C08965=1019.841,-8.472,-102.051,166.453,52.235,159.485
C08966=1019.835,-8.722,-102.038,166.450,52.240,159.486
C08967=1019.829,-8.971,-102.024,166.447,52.245,159.486
C08968=1019.824,-9.221,-102.010,166.445,52.250,159.487
C08969=1019.818,-9.471,-101.998,166.442,52.256,159.487
C08970=1019.812,-9.720,-101.985,166.439,52.261,159.487
C08971=1019.806,-9.970,-101.971,166.436,52.266,159.488
C08972=1019.801,-10.219,-101.959,166.434,52.272,159.489
C08973=1019.796,-10.469,-101.945,166.431,52.277,159.489
C08974=1019.789,-10.718,-101.932,166.428,52.283,159.489
C08975=1019.784,-10.968,-101.918,166.425,52.288,159.490
C08976=1019.778,-11.218,-101.906,166.423,52.293,159.490
C08977=1019.772,-11.467,-101.892,166.420,52.298,159.491
C08978=1019.767,-11.717,-101.879,166.417,52.304,159.491
C08979=1019.760,-11.966,-101.866,166.414,52.309,159.491
C08980=1019.756,-12.216,-101.853,166.412,52.314,159.492
C08981=1019.750,-12.465,-101.840,166.408,52.319,159.492
C08982=1019.745,-12.715,-101.827,166.405,52.324,159.493
C08983=1019.738,-12.965,-101.814,166.403,52.331,159.493
C08984=1019.732,-13.215,-101.801,166.401,52.335,159.494
C08985=1019.727,-13.464,-101.787,166.398,52.341,159.494
C08986=1019.722,-13.713,-101.775,166.395,52.346,159.495
C08987=1019.716,-13.963,-101.761,166.393,52.351,159.495
C08988=1019.710,-14.213,-101.749,166.389,52.356,159.496
C08989=1019.704,-14.463,-101.736,166.386,52.362,159.496
C08990=1019.699,-14.712,-101.722,166.383,52.367,159.496
C08991=1019.694,-14.961,-101.710,166.381,52.372,159.497
C08992=1019.688,-15.211,-101.696,166.378,52.377,159.497
C08993=1019.682,-15.461,-101.684,166.375,52.383,159.498
C08994=1019.676,-15.710,-101.670,166.373,52.388,159.498
C08995=1019.671,-15.960,-101.657,166.370,52.393,159.499
C08996=1019.665,-16.209,-101.645,166.367,52.398,159.499
C08997=1019.660,-16.459,-101.632,166.364,52.404,159.499
C08998=1019.653,-16.709,-101.619,166.361,52.409,159.500
C08999=1019.647,-16.959,-101.607,166.359,52.414,159.500
C09000=1019.642,-17.209,-101.593,166.356,52.419,159.501
C09001=1019.637,-17.457,-101.580,166.353,52.425,159.501
C09002=1019.631,-17.707,-101.568,166.350,52.431,159.502
C09003=1019.625,-17.957,-101.555,166.347,52.436,159.502
C09004=1019.619,-18.207,-101.543,166.345,52.441,159.503
C09005=1019.614,-18.456,-101.531,166.342,52.446,159.503
C09006=1019.607,-18.705,-101.517,166.339,52.452,159.503
C09007=1019.602,-18.956,-101.504,166.336,52.457,159.504
C09008=1019.596,-19.205,-101.492,166.334,52.462,159.504
C09009=1019.591,-19.455,-101.479,166.331,52.467,159.505
C09010=1019.585,-19.705,-101.467,166.328,52.473,159.505
C09011=1019.579,-19.954,-101.454,166.325,52.479,159.506
C09012=1019.574,-20.203,-101.441,166.322,52.484,159.506
C09013=1019.568,-20.453,-101.429,166.320,52.489,159.507
C09014=1019.562,-20.703,-101.416,166.317,52.494,159.507
C09015=1019.556,-20.981,-101.402,166.314,52.500,159.507
C09016=1019.550,-21.259,-101.388,166.310,52.506,159.508
C09017=1019.543,-21.539,-101.373,166.307,52.512,159.509
C09018=1019.537,-21.817,-101.360,166.304,52.518,159.509
C09019=1019.531,-22.067,-101.347,166.301,52.523,159.509
C09020=1019.525,-22.316,-101.335,166.298,52.528,159.510
C09021=1019.520,-22.566,-101.322,166.295,52.534,159.510
C09022=1019.514,-22.816,-101.309,166.293,52.539,159.511
C09023=1019.509,-23.065,-101.297,166.290,52.544,159.511
C09024=1019.503,-23.315,-101.284,166.287,52.549,159.511
C09025=1019.497,-23.565,-101.271,166.284,52.555,159.512
C09026=1019.492,-23.814,-101.259,166.281,52.560,159.512
C09027=1019.486,-24.064,-101.246,166.279,52.565,159.513
C09028=1019.480,-24.314,-101.234,166.276,52.570,159.513
C09029=1019.475,-24.563,-101.221,166.273,52.576,159.514
C09030=1019.469,-24.813,-101.209,166.271,52.581,159.514
C09031=1019.464,-25.062,-101.196,166.268,52.586,159.514
C09032=1019.458,-25.312,-101.184,166.265,52.591,159.515
C09033=1019.452,-25.562,-101.171,166.262,52.597,159.515
C09034=1019.447,-25.811,-101.159,166.260,52.602,159.516
C09035=1019.441,-26.061,-101.147,166.256,52.606,159.516
C09036=1019.436,-26.310,-101.134,166.253,52.612,159.516
C09037=1019.430,-26.560,-101.122,166.250,52.617,159.517
C09038=1019.425,-26.810,-101.109,166.248,52.622,159.517
C09039=1019.419,-27.059,-101.096,166.245,52.628,159.518
C09040=1019.413,-27.309,-101.084,166.242,52.633,159.518
C09041=1019.408,-27.558,-101.072,166.239,52.638,159.518
C09042=1019.402,-27.808,-101.059,166.237,52.643,159.519
C09043=1019.397,-28.059,-101.047,166.234,52.649,159.519
C09044=1019.391,-28.308,-101.035,166.231,52.654,159.520
C09045=1019.385,-28.558,-101.023,166.228,52.659,159.520
C09046=1019.379,-28.807,-101.011,166.225,52.665,159.520
C09047=1019.373,-29.057,-100.998,166.223,52.670,159.521
C09048=1019.368,-29.306,-100.986,166.220,52.675,159.521
C09049=1019.363,-29.556,-100.974,166.217,52.680,159.522
C09050=1019.357,-29.806,-100.962,166.214,52.686,159.522
C09051=1019.351,-30.055,-100.950,166.211,52.691,159.523
C09052=1019.345,-30.305,-100.938,166.208,52.697,159.523
C09053=1019.340,-30.555,-100.926,166.206,52.702,159.523
C09054=1019.334,-30.805,-100.914,166.203,52.707,159.524
C09055=1019.328,-31.054,-100.902,166.200,52.712,159.524
C09056=1019.323,-31.304,-100.889,166.197,52.718,159.525
C09057=1019.317,-31.553,-100.878,166.193,52.723,159.525
C09058=1019.311,-31.803,-100.866,166.191,52.728,159.526
C09059=1019.306,-32.052,-100.853,166.188,52.733,159.526
C09060=1019.300,-32.302,-100.841,166.185,52.739,159.526
C09061=1019.295,-32.552,-100.829,166.182,52.744,159.527
C09062=1019.289,-32.802,-100.817,166.179,52.749,159.527
C09063=1019.283,-33.051,-100.805,166.177,52.755,159.528
C09064=1019.277,-33.301,-100.793,166.174,52.760,159.528
C09065=1019.272,-33.550,-100.781,166.171,52.765,159.528
C09066=1019.266,-33.800,-100.769,166.168,52.771,159.529
C09067=1019.261,-34.050,-100.757,166.165,52.775,159.529
C09068=1019.255,-34.299,-100.746,166.163,52.780,159.529
C09069=1019.249,-34.549,-100.733,166.160,52.786,159.530
C09070=1019.244,-34.799,-100.722,166.157,52.791,159.530
C09071=1019.238,-35.049,-100.709,166.154,52.796,159.531
C09072=1019.233,-35.298,-100.697,166.151,52.802,159.531
C09073=1019.228,-35.548,-100.685,166.149,52.807,159.531
C09074=1019.221,-35.797,-100.673,166.146,52.812,159.532
C09075=1019.216,-36.047,-100.662,166.143,52.818,159.532
C09076=1019.210,-36.297,-100.649,166.140,52.823,159.533
C09077=1019.205,-36.546,-100.637,166.136,52.828,159.533
C09078=1019.200,-36.796,-100.626,166.134,52.833,159.533
C09079=1019.193,-37.074,-100.612,166.130,52.839,159.534
C09080=1019.187,-37.352,-100.599,166.127,52.845,159.534
C09081=1019.181,-37.629,-100.586,166.124,52.850,159.535
C09082=1019.175,-37.908,-100.573,166.121,52.856,159.535
C09083=1019.169,-38.157,-100.560,166.119,52.861,159.536
C09084=1019.163,-38.406,-100.549,166.116,52.867,159.536
C09085=1019.158,-38.656,-100.537,166.112,52.871,159.536
C09086=1019.152,-38.905,-100.525,166.109,52.877,159.536
C09087=1019.147,-39.155,-100.513,166.107,52.882,159.537
C09088=1019.141,-39.405,-100.501,166.104,52.887,159.537
C09089=1019.136,-39.655,-100.490,166.101,52.893,159.538
C09090=1019.131,-39.904,-100.478,166.098,52.898,159.538
C09091=1019.124,-40.154,-100.466,166.095,52.903,159.539
C09092=1019.119,-40.404,-100.455,166.092,52.909,159.539
C09093=1019.113,-40.653,-100.444,166.089,52.914,159.539
C09094=1019.107,-40.903,-100.432,166.087,52.919,159.540
C09095=1019.102,-41.153,-100.421,166.084,52.925,159.540
C09096=1019.097,-41.402,-100.409,166.081,52.930,159.541
C09097=1019.090,-41.652,-100.397,166.078,52.935,159.541
C09098=1019.085,-41.902,-100.386,166.075,52.941,159.541
C09099=1019.079,-42.151,-100.375,166.072,52.946,159.542
C09100=1019.073,-42.401,-100.362,166.069,52.951,159.542
C09101=1019.068,-42.651,-100.351,166.066,52.956,159.542
C09102=1019.063,-42.900,-100.340,166.064,52.961,159.543
C09103=1019.057,-43.150,-100.328,166.061,52.967,159.543
C09104=1019.051,-43.400,-100.317,166.058,52.972,159.544
C09105=1019.046,-43.650,-100.305,166.055,52.978,159.544
C09106=1019.040,-43.899,-100.294,166.052,52.983,159.544
C09107=1019.034,-44.149,-100.282,166.049,52.988,159.545
C09108=1019.029,-44.399,-100.271,166.047,52.993,159.545
C09109=1019.024,-44.648,-100.259,166.044,52.999,159.546
C09110=1019.018,-44.898,-100.248,166.041,53.004,159.546
C09111=1019.012,-45.148,-100.236,166.037,53.009,159.546
C09112=1019.006,-45.397,-100.225,166.034,53.014,159.546
C09113=1019.001,-45.647,-100.214,166.031,53.020,159.547
C09114=1018.995,-45.896,-100.203,166.028,53.025,159.547
C09115=1018.990,-46.146,-100.190,166.026,53.030,159.548
C09116=1018.984,-46.396,-100.179,166.023,53.036,159.548
C09117=1018.979,-46.646,-100.168,166.020,53.041,159.549
C09118=1018.973,-46.895,-100.157,166.017,53.046,159.549
C09119=1018.968,-47.145,-100.145,166.014,53.051,159.549
C09120=1018.962,-47.394,-100.135,166.011,53.056,159.549
C09121=1018.956,-47.644,-100.122,166.009,53.061,159.550
C09122=1018.951,-47.894,-100.111,166.006,53.067,159.550
C09123=1018.946,-48.144,-100.100,166.003,53.072,159.551
C09124=1018.940,-48.393,-100.089,165.999,53.077,159.551
C09125=1018.935,-48.643,-100.077,165.996,53.082,159.551
C09126=1018.930,-48.893,-100.066,165.994,53.087,159.552
C09127=1018.924,-49.142,-100.055,165.991,53.093,159.552
C09128=1018.919,-49.393,-100.043,165.988,53.098,159.552
C09129=1018.913,-49.642,-100.031,165.985,53.103,159.553
C09130=1018.908,-49.891,-100.020,165.982,53.108,159.553
C09131=1018.902,-50.141,-100.009,165.979,53.114,159.553
C09132=1018.897,-50.391,-99.998,165.977,53.119,159.554
C09133=1018.891,-50.640,-99.987,165.974,53.124,159.554
C09134=1018.886,-50.890,-99.975,165.970,53.129,159.554
C09135=1018.880,-51.140,-99.964,165.967,53.134,159.555
C09136=1018.874,-51.390,-99.953,165.964,53.140,159.555
C09137=1018.868,-51.639,-99.942,165.961,53.145,159.556
C09138=1018.863,-51.889,-99.932,165.958,53.151,159.556
C09139=1018.857,-52.139,-99.921,165.955,53.156,159.556
C09140=1018.851,-52.388,-99.910,165.952,53.161,159.557
C09141=1018.846,-52.638,-99.899,165.949,53.167,159.557
C09142=1018.841,-52.887,-99.888,165.946,53.172,159.557
C09143=1018.834,-53.165,-99.876,165.944,53.178,159.558
C09144=1018.827,-53.444,-99.864,165.940,53.185,159.558
C09145=1018.821,-53.722,-99.852,165.937,53.190,159.559
C09146=1018.815,-54.000,-99.840,165.934,53.197,159.559
C09147=1018.809,-54.250,-99.829,165.931,53.202,159.560
///RCONF 1,0,0,1,0,0,0,0,0,0,0,0,0,0,0,0,0,0,0,0,0,0,0,0
C09148=1018.804,-54.499,-99.818,165.928,53.208,159.560
C09149=1018.798,-54.749,-99.808,165.925,53.213,159.560
C09150=1018.792,-54.999,-99.797,165.922,53.219,159.561
C09151=1018.787,-55.248,-99.786,165.919,53.224,159.561
C09152=1018.782,-55.498,-99.775,165.916,53.229,159.562
C09153=1018.776,-55.748,-99.765,165.914,53.235,159.562
C09154=1018.770,-55.998,-99.754,165.911,53.240,159.562
C09155=1018.765,-56.247,-99.743,165.908,53.245,159.563
C09156=1018.759,-56.497,-99.732,165.905,53.251,159.563
C09157=1018.754,-56.747,-99.722,165.901,53.256,159.563
C09158=1018.748,-56.996,-99.711,165.898,53.261,159.564
C09159=1018.742,-57.246,-99.700,165.895,53.266,159.564
C09160=1018.737,-57.496,-99.690,165.892,53.272,159.564
C09161=1018.731,-57.745,-99.679,165.889,53.277,159.565
C09162=1018.726,-57.995,-99.668,165.886,53.283,159.565
C09163=1018.720,-58.245,-99.657,165.883,53.288,159.566
C09164=1018.715,-58.495,-99.647,165.880,53.294,159.566
C09165=1018.709,-58.744,-99.636,165.877,53.299,159.566
C09166=1018.704,-58.994,-99.626,165.874,53.304,159.567
C09167=1018.698,-59.244,-99.615,165.871,53.310,159.567
C09168=1018.692,-59.493,-99.604,165.868,53.315,159.567
C09169=1018.687,-59.743,-99.594,165.865,53.320,159.568
C09170=1018.681,-59.993,-99.583,165.863,53.325,159.568
C09171=1018.675,-60.243,-99.573,165.860,53.331,159.568
C09172=1018.670,-60.493,-99.562,165.857,53.336,159.569
C09173=1018.665,-60.741,-99.551,165.854,53.341,159.569
C09174=1018.660,-60.992,-99.540,165.851,53.347,159.570
C09175=1018.654,-61.241,-99.530,165.848,53.352,159.570
C09176=1018.649,-61.491,-99.519,165.845,53.357,159.570
C09177=1018.643,-61.741,-99.509,165.842,53.363,159.570
C09178=1018.637,-61.990,-99.498,165.839,53.368,159.571
C09179=1018.632,-62.240,-99.487,165.836,53.373,159.571
C09180=1018.626,-62.490,-99.477,165.833,53.379,159.571
C09181=1018.621,-62.740,-99.466,165.830,53.384,159.572
C09182=1018.615,-62.989,-99.456,165.827,53.389,159.572
C09183=1018.610,-63.239,-99.446,165.824,53.394,159.573
C09184=1018.604,-63.488,-99.435,165.821,53.400,159.573
C09185=1018.599,-63.739,-99.425,165.818,53.405,159.573
C09186=1018.593,-63.988,-99.414,165.815,53.410,159.574
C09187=1018.588,-64.238,-99.404,165.812,53.416,159.574
C09188=1018.583,-64.488,-99.392,165.809,53.421,159.574
C09189=1018.578,-64.737,-99.382,165.806,53.426,159.574
C09190=1018.572,-64.987,-99.372,165.803,53.432,159.575
C09191=1018.567,-65.237,-99.361,165.800,53.437,159.575
C09192=1018.561,-65.487,-99.351,165.798,53.441,159.576
C09193=1018.556,-65.737,-99.340,165.795,53.447,159.576
C09194=1018.551,-65.986,-99.331,165.792,53.452,159.576
C09195=1018.545,-66.235,-99.320,165.789,53.458,159.577
C09196=1018.540,-66.486,-99.310,165.785,53.462,159.577
C09197=1018.534,-66.735,-99.299,165.782,53.468,159.577
C09198=1018.528,-66.985,-99.288,165.779,53.473,159.577
C09199=1018.524,-67.235,-99.279,165.776,53.479,159.578
C09200=1018.518,-67.484,-99.268,165.774,53.483,159.578
C09201=1018.512,-67.734,-99.258,165.771,53.489,159.579
C09202=1018.507,-67.984,-99.247,165.768,53.494,159.579
C09203=1018.502,-68.233,-99.237,165.765,53.499,159.579
C09204=1018.496,-68.483,-99.227,165.762,53.504,159.579
C09205=1018.491,-68.733,-99.215,165.759,53.510,159.580
C09206=1018.486,-68.983,-99.205,165.756,53.515,159.580
C09207=1018.479,-69.286,-99.193,165.752,53.521,159.580
C09208=1018.473,-69.590,-99.180,165.748,53.528,159.581
C09209=1018.466,-69.893,-99.168,165.746,53.534,159.581
C09210=1018.460,-70.196,-99.156,165.742,53.540,159.582
C09211=1018.455,-70.446,-99.145,165.739,53.545,159.582
C09212=1018.449,-70.696,-99.134,165.736,53.551,159.582
C09213=1018.445,-70.945,-99.125,165.732,53.555,159.582
C09214=1018.439,-71.196,-99.114,165.729,53.561,159.583
C09215=1018.433,-71.445,-99.104,165.726,53.566,159.583
C09216=1018.429,-71.694,-99.094,165.724,53.571,159.583
C09217=1018.423,-71.945,-99.084,165.721,53.576,159.584
C09218=1018.418,-72.195,-99.073,165.718,53.582,159.584
C09219=1018.413,-72.443,-99.063,165.715,53.586,159.584
C09220=1018.407,-72.694,-99.053,165.712,53.592,159.585
C09221=1018.402,-72.944,-99.043,165.708,53.597,159.585
C09222=1018.397,-73.193,-99.033,165.706,53.602,159.585
C09223=1018.391,-73.443,-99.022,165.703,53.607,159.586
C09224=1018.386,-73.693,-99.012,165.700,53.612,159.586
C09225=1018.381,-73.942,-99.002,165.697,53.617,159.586
C09226=1018.375,-74.192,-98.992,165.693,53.622,159.586
C09227=1018.370,-74.442,-98.982,165.691,53.628,159.587
C09228=1018.365,-74.692,-98.972,165.688,53.633,159.587
C09229=1018.360,-74.942,-98.962,165.685,53.639,159.587
C09230=1018.354,-75.191,-98.953,165.682,53.643,159.588
C09231=1018.349,-75.441,-98.942,165.679,53.648,159.588
C09232=1018.343,-75.691,-98.932,165.676,53.654,159.588
C09233=1018.338,-75.941,-98.922,165.673,53.659,159.589
C09234=1018.332,-76.190,-98.913,165.670,53.665,159.589
C09235=1018.327,-76.440,-98.903,165.667,53.670,159.589
C09236=1018.322,-76.690,-98.893,165.664,53.675,159.590
C09237=1018.316,-76.940,-98.883,165.661,53.681,159.590
C09238=1018.311,-77.189,-98.874,165.658,53.686,159.590
C09239=1018.306,-77.439,-98.863,165.655,53.691,159.590
C09240=1018.301,-77.689,-98.854,165.652,53.696,159.591
C09241=1018.295,-77.938,-98.844,165.649,53.702,159.591
C09242=1018.290,-78.188,-98.834,165.646,53.707,159.591
C09243=1018.285,-78.426,-98.825,165.643,53.712,159.592
C09244=1018.280,-78.663,-98.816,165.641,53.717,159.592
C09245=1018.275,-78.901,-98.806,165.637,53.722,159.592
C09246=1018.269,-79.139,-98.797,165.634,53.727,159.593
C09247=1018.264,-79.376,-98.788,165.632,53.732,159.593
C09248=1018.259,-79.614,-98.779,165.629,53.737,159.593
C09249=1018.254,-79.851,-98.769,165.625,53.742,159.593
C09250=1018.249,-80.089,-98.759,165.624,53.747,159.594
C09251=1018.244,-80.339,-98.751,165.620,53.752,159.594
C09252=1018.239,-80.589,-98.741,165.617,53.757,159.594
C09253=1018.233,-80.838,-98.731,165.614,53.763,159.595
C09254=1018.228,-81.088,-98.721,165.611,53.768,159.595
C09255=1018.222,-81.338,-98.713,165.608,53.774,159.595
C09256=1018.217,-81.588,-98.703,165.605,53.779,159.596
C09257=1018.211,-81.837,-98.693,165.602,53.785,159.596
C09258=1018.205,-82.088,-98.685,165.599,53.790,159.597
C09259=1018.201,-82.337,-98.675,165.597,53.796,159.597
C09260=1018.194,-82.587,-98.665,165.593,53.801,159.597
C09261=1018.190,-82.837,-98.656,165.590,53.806,159.597
C09262=1018.184,-83.087,-98.647,165.587,53.812,159.598
C09263=1018.179,-83.336,-98.637,165.584,53.817,159.598
C09264=1018.173,-83.586,-98.628,165.581,53.823,159.598
C09265=1018.168,-83.836,-98.618,165.578,53.828,159.599
C09266=1018.163,-84.085,-98.609,165.575,53.834,159.599
C09267=1018.157,-84.335,-98.600,165.572,53.838,159.599
C09268=1018.152,-84.585,-98.590,165.569,53.844,159.600
C09269=1018.146,-84.835,-98.581,165.566,53.849,159.600
C09270=1018.141,-85.085,-98.572,165.563,53.855,159.600
C09271=1018.135,-85.366,-98.561,165.559,53.861,159.600
C09272=1018.129,-85.647,-98.551,165.556,53.867,159.601
C09273=1018.122,-85.928,-98.540,165.553,53.873,159.601
C09274=1018.117,-86.209,-98.530,165.549,53.879,159.602
C09275=1018.111,-86.459,-98.521,165.546,53.884,159.602
C09276=1018.106,-86.709,-98.511,165.543,53.890,159.602
C09277=1018.101,-86.958,-98.503,165.540,53.895,159.603
C09278=1018.096,-87.208,-98.492,165.537,53.901,159.603
C09279=1018.090,-87.458,-98.484,165.534,53.906,159.603
C09280=1018.086,-87.708,-98.474,165.531,53.911,159.603
C09281=1018.080,-87.958,-98.465,165.528,53.917,159.604
C09282=1018.075,-88.207,-98.455,165.525,53.922,159.604
C09283=1018.070,-88.457,-98.447,165.522,53.928,159.604
C09284=1018.063,-88.707,-98.437,165.518,53.932,159.605
C09285=1018.059,-88.957,-98.428,165.515,53.938,159.605
C09286=1018.053,-89.206,-98.419,165.513,53.943,159.605
C09287=1018.048,-89.457,-98.410,165.510,53.949,159.606
C09288=1018.043,-89.706,-98.400,165.506,53.954,159.606
C09289=1018.037,-89.956,-98.392,165.503,53.959,159.606
C09290=1018.032,-90.206,-98.382,165.500,53.965,159.606
C09291=1018.027,-90.455,-98.373,165.498,53.969,159.607
C09292=1018.022,-90.705,-98.364,165.495,53.975,159.607
C09293=1018.017,-90.954,-98.355,165.492,53.980,159.607
C09294=1018.012,-91.205,-98.346,165.489,53.986,159.608
C09295=1018.006,-91.454,-98.336,165.486,53.990,159.608
C09296=1018.001,-91.704,-98.328,165.483,53.996,159.608
C09297=1017.996,-91.953,-98.318,165.480,54.001,159.609
C09298=1017.990,-92.204,-98.309,165.477,54.006,159.609
C09299=1017.985,-92.454,-98.300,165.474,54.012,159.609
C09300=1017.980,-92.703,-98.291,165.471,54.017,159.609
C09301=1017.975,-92.953,-98.283,165.467,54.022,159.609
C09302=1017.970,-93.203,-98.273,165.464,54.028,159.610
C09303=1017.964,-93.453,-98.264,165.461,54.033,159.610
C09304=1017.959,-93.703,-98.255,165.458,54.038,159.610
C09305=1017.954,-93.952,-98.246,165.455,54.043,159.611
C09306=1017.949,-94.201,-98.237,165.452,54.049,159.611
C09307=1017.944,-94.451,-98.228,165.450,54.053,159.611
C09308=1017.938,-94.702,-98.219,165.447,54.059,159.612
C09309=1017.933,-94.951,-98.209,165.444,54.064,159.612
C09310=1017.928,-95.201,-98.201,165.441,54.069,159.612
C09311=1017.923,-95.451,-98.192,165.438,54.075,159.612
C09312=1017.918,-95.701,-98.183,165.434,54.080,159.613
C09313=1017.913,-95.950,-98.174,165.431,54.085,159.613
C09314=1017.908,-96.200,-98.165,165.428,54.091,159.613
C09315=1017.902,-96.450,-98.156,165.425,54.095,159.613
C09316=1017.897,-96.700,-98.148,165.422,54.101,159.614
C09317=1017.892,-96.949,-98.138,165.420,54.105,159.614
C09318=1017.887,-97.199,-98.129,165.417,54.111,159.614
C09319=1017.882,-97.449,-98.120,165.414,54.116,159.615
C09320=1017.877,-97.699,-98.112,165.411,54.121,159.615
C09321=1017.871,-97.949,-98.103,165.408,54.127,159.615
C09322=1017.867,-98.199,-98.094,165.405,54.132,159.615
C09323=1017.861,-98.448,-98.085,165.401,54.137,159.616
C09324=1017.856,-98.698,-98.076,165.398,54.143,159.616
C09325=1017.851,-98.948,-98.068,165.395,54.148,159.616
C09326=1017.845,-99.197,-98.059,165.393,54.154,159.617
C09327=1017.840,-99.447,-98.051,165.390,54.159,159.617
C09328=1017.835,-99.697,-98.042,165.386,54.164,159.617
C09329=1017.830,-99.947,-98.034,165.383,54.170,159.617
C09330=1017.825,-100.197,-98.025,165.380,54.175,159.618
C09331=1017.820,-100.446,-98.016,165.378,54.181,159.618
C09332=1017.815,-100.696,-98.008,165.374,54.186,159.618
C09333=1017.809,-100.946,-97.999,165.371,54.191,159.619
C09334=1017.803,-101.196,-97.990,165.368,54.197,159.619
C09335=1017.798,-101.479,-97.981,165.364,54.203,159.619
C09336=1017.792,-101.763,-97.971,165.362,54.209,159.620
C09337=1017.786,-102.046,-97.961,165.358,54.215,159.620
C09338=1017.780,-102.329,-97.952,165.354,54.221,159.620
C09339=1017.776,-102.579,-97.943,165.351,54.226,159.620
C09340=1017.771,-102.829,-97.935,165.348,54.232,159.621
C09341=1017.765,-103.079,-97.927,165.346,54.236,159.621
C09342=1017.760,-103.328,-97.918,165.343,54.242,159.621
C09343=1017.755,-103.578,-97.910,165.340,54.247,159.622
C09344=1017.750,-103.828,-97.901,165.337,54.252,159.622
C09345=1017.744,-104.078,-97.893,165.334,54.258,159.622
C09346=1017.739,-104.327,-97.884,165.331,54.263,159.622
C09347=1017.734,-104.577,-97.876,165.328,54.269,159.623
C09348=1017.728,-104.827,-97.867,165.324,54.274,159.623
C09349=1017.723,-105.077,-97.860,165.322,54.279,159.623
C09350=1017.718,-105.327,-97.851,165.319,54.285,159.624
C09351=1017.714,-105.577,-97.842,165.315,54.289,159.624
C09352=1017.708,-105.826,-97.834,165.312,54.295,159.624
C09353=1017.703,-106.076,-97.825,165.309,54.301,159.624
C09354=1017.698,-106.327,-97.817,165.306,54.305,159.624
C09355=1017.693,-106.576,-97.809,165.303,54.311,159.625
C09356=1017.688,-106.826,-97.800,165.300,54.316,159.625
C09357=1017.682,-107.076,-97.792,165.297,54.321,159.625
C09358=1017.678,-107.325,-97.784,165.294,54.327,159.626
C09359=1017.673,-107.575,-97.776,165.291,54.332,159.626
C09360=1017.668,-107.825,-97.768,165.288,54.337,159.626
C09361=1017.662,-108.074,-97.759,165.285,54.343,159.626
C09362=1017.657,-108.325,-97.751,165.282,54.348,159.627
C09363=1017.652,-108.575,-97.743,165.279,54.354,159.627
C09364=1017.647,-108.824,-97.734,165.276,54.359,159.627
C09365=1017.641,-109.074,-97.727,165.273,54.364,159.627
C09366=1017.636,-109.324,-97.719,165.270,54.370,159.628
C09367=1017.631,-109.573,-97.711,165.267,54.375,159.628
C09368=1017.626,-109.823,-97.703,165.264,54.380,159.628
C09369=1017.621,-110.073,-97.694,165.261,54.386,159.629
C09370=1017.616,-110.323,-97.687,165.258,54.391,159.629
C09371=1017.611,-110.573,-97.678,165.254,54.396,159.629
C09372=1017.605,-110.823,-97.670,165.253,54.401,159.629
C09373=1017.601,-111.072,-97.662,165.250,54.407,159.630
C09374=1017.595,-111.322,-97.654,165.247,54.413,159.630
C09375=1017.590,-111.572,-97.647,165.243,54.417,159.630
C09376=1017.585,-111.822,-97.638,165.240,54.423,159.631
C09377=1017.580,-112.072,-97.630,165.238,54.428,159.631
C09378=1017.575,-112.321,-97.622,165.234,54.433,159.631
C09379=1017.570,-112.571,-97.614,165.231,54.439,159.631
C09380=1017.565,-112.821,-97.606,165.228,54.444,159.632
C09381=1017.560,-113.071,-97.597,165.225,54.449,159.632
C09382=1017.555,-113.321,-97.590,165.222,54.455,159.632
C09383=1017.549,-113.570,-97.582,165.219,54.460,159.632
C09384=1017.544,-113.820,-97.574,165.216,54.465,159.633
C09385=1017.539,-114.070,-97.566,165.213,54.471,159.633
C09386=1017.534,-114.320,-97.558,165.210,54.476,159.633
C09387=1017.530,-114.569,-97.550,165.207,54.481,159.633
C09388=1017.525,-114.820,-97.542,165.204,54.487,159.634
C09389=1017.519,-115.070,-97.535,165.201,54.492,159.634
C09390=1017.514,-115.319,-97.527,165.198,54.497,159.634
C09391=1017.509,-115.569,-97.519,165.195,54.503,159.634
C09392=1017.504,-115.819,-97.511,165.192,54.508,159.635
C09393=1017.498,-116.069,-97.503,165.188,54.513,159.635
C09394=1017.494,-116.319,-97.496,165.186,54.519,159.635
C09395=1017.489,-116.568,-97.488,165.183,54.524,159.636
C09396=1017.484,-116.819,-97.480,165.181,54.530,159.636
C09397=1017.479,-117.068,-97.472,165.177,54.534,159.636
C09398=1017.473,-117.318,-97.465,165.175,54.540,159.636
C09399=1017.468,-117.601,-97.456,165.171,54.546,159.637
C09400=1017.462,-117.885,-97.447,165.167,54.553,159.637
C09401=1017.457,-118.168,-97.438,165.164,54.558,159.637
C09402=1017.451,-118.451,-97.429,165.160,54.564,159.637
C09403=1017.446,-118.701,-97.422,165.157,54.570,159.638
C09404=1017.440,-118.951,-97.414,165.155,54.575,159.638
C09405=1017.435,-119.200,-97.406,165.151,54.580,159.638
C09406=1017.430,-119.451,-97.399,165.148,54.586,159.639
C09407=1017.425,-119.700,-97.392,165.145,54.591,159.639
C09408=1017.420,-119.950,-97.384,165.142,54.596,159.639
C09409=1017.415,-120.201,-97.376,165.139,54.602,159.639
C09410=1017.411,-120.450,-97.368,165.137,54.607,159.640
C09411=1017.405,-120.700,-97.361,165.134,54.612,159.640
C09412=1017.400,-120.950,-97.353,165.131,54.618,159.640
C09413=1017.396,-121.200,-97.346,165.128,54.623,159.641
C09414=1017.390,-121.450,-97.339,165.125,54.628,159.641
C09415=1017.385,-121.699,-97.330,165.122,54.634,159.641
C09416=1017.380,-121.949,-97.323,165.119,54.639,159.641
C09417=1017.375,-122.198,-97.316,165.116,54.644,159.641
C09418=1017.370,-122.449,-97.308,165.113,54.650,159.642
C09419=1017.365,-122.699,-97.300,165.110,54.655,159.642
C09420=1017.360,-122.948,-97.294,165.107,54.660,159.642
C09421=1017.355,-123.199,-97.286,165.104,54.666,159.643
C09422=1017.350,-123.447,-97.278,165.100,54.670,159.643
C09423=1017.345,-123.698,-97.270,165.098,54.676,159.643
C09424=1017.341,-123.947,-97.263,165.095,54.682,159.643
C09425=1017.335,-124.197,-97.256,165.092,54.686,159.644
C09426=1017.331,-124.447,-97.249,165.090,54.692,159.644
C09427=1017.326,-124.697,-97.241,165.087,54.697,159.644
C09428=1017.321,-124.947,-97.234,165.083,54.702,159.644
C09429=1017.316,-125.197,-97.226,165.080,54.708,159.645
C09430=1017.311,-125.446,-97.219,165.078,54.713,159.645
C09431=1017.306,-125.697,-97.212,165.074,54.718,159.645
C09432=1017.300,-125.946,-97.205,165.071,54.724,159.645
C09433=1017.296,-126.196,-97.197,165.068,54.729,159.646
C09434=1017.290,-126.446,-97.190,165.065,54.734,159.646
C09435=1017.285,-126.696,-97.182,165.062,54.740,159.646
C09436=1017.280,-126.945,-97.176,165.059,54.746,159.646
C09437=1017.275,-127.196,-97.168,165.056,54.750,159.646
C09438=1017.270,-127.445,-97.161,165.053,54.756,159.647
C09439=1017.266,-127.694,-97.154,165.050,54.762,159.647
C09440=1017.260,-127.944,-97.146,165.047,54.766,159.647
C09441=1017.256,-128.194,-97.139,165.045,54.772,159.648
C09442=1017.252,-128.444,-97.132,165.042,54.777,159.648
C09443=1017.248,-128.693,-97.123,165.039,54.780,159.648
C09444=1017.244,-128.942,-97.114,165.036,54.784,159.648
C09445=1017.240,-129.193,-97.105,165.033,54.787,159.648
C09446=1017.237,-129.442,-97.094,165.031,54.790,159.648
C09447=1017.235,-129.692,-97.083,165.028,54.792,159.647
C09448=1017.233,-129.941,-97.072,165.026,54.793,159.647
C09449=1017.231,-130.191,-97.060,165.023,54.794,159.646
C09450=1017.230,-130.441,-97.047,165.021,54.794,159.646
C09451=1017.229,-130.690,-97.034,165.019,54.794,159.646
C09452=1017.229,-130.940,-97.020,165.017,54.793,159.645
C09453=1017.229,-131.190,-97.006,165.014,54.791,159.644
C09454=1017.229,-131.439,-96.991,165.012,54.789,159.643
C09455=1017.230,-131.689,-96.975,165.010,54.787,159.642
C09456=1017.231,-131.938,-96.959,165.008,54.784,159.641
C09457=1017.233,-132.189,-96.943,165.006,54.780,159.640
C09458=1017.235,-132.438,-96.924,165.005,54.776,159.639
C09459=1017.237,-132.688,-96.907,165.003,54.771,159.638
C09460=1017.240,-132.938,-96.888,165.000,54.766,159.636
C09461=1017.243,-133.188,-96.869,164.999,54.760,159.635
C09462=1017.247,-133.437,-96.850,164.997,54.753,159.634
C09463=1016.989,-133.463,-97.235,164.957,55.109,159.686
C09464=1016.985,-133.214,-97.254,164.959,55.115,159.688
C09465=1016.982,-132.964,-97.273,164.960,55.121,159.689
C09466=1016.980,-132.715,-97.292,164.962,55.126,159.691
C09467=1016.977,-132.464,-97.310,164.964,55.131,159.692
C09468=1016.975,-132.215,-97.327,164.966,55.135,159.693
C09469=1016.974,-131.965,-97.344,164.968,55.139,159.694
C09470=1016.972,-131.715,-97.361,164.970,55.142,159.695
C09471=1016.971,-131.466,-97.377,164.972,55.145,159.696
C09472=1016.971,-131.216,-97.392,164.974,55.147,159.697
C09473=1016.971,-130.967,-97.406,164.976,55.148,159.698
C09474=1016.971,-130.717,-97.420,164.979,55.149,159.699
C09475=1016.972,-130.467,-97.433,164.980,55.149,159.699
C09476=1016.974,-130.218,-97.445,164.983,55.149,159.700
C09477=1016.975,-129.968,-97.457,164.985,55.148,159.700
C09478=1016.977,-129.718,-97.468,164.988,55.146,159.700
C09479=1016.979,-129.468,-97.480,164.991,55.144,159.701
C09480=1016.982,-129.219,-97.490,164.993,55.142,159.701
C09481=1016.985,-128.969,-97.500,164.996,55.139,159.701
C09482=1016.989,-128.719,-97.509,164.999,55.135,159.701
C09483=1016.993,-128.470,-97.517,165.002,55.131,159.701
C09484=1016.998,-128.220,-97.525,165.004,55.127,159.701
C09485=1017.002,-127.971,-97.532,165.007,55.121,159.700
C09486=1017.007,-127.722,-97.539,165.010,55.116,159.700
C09487=1017.012,-127.471,-97.547,165.013,55.111,159.700
C09488=1017.017,-127.222,-97.554,165.016,55.105,159.699
C09489=1017.022,-126.972,-97.561,165.018,55.099,159.699
C09490=1017.027,-126.722,-97.568,165.022,55.094,159.699
C09491=1017.032,-126.473,-97.576,165.025,55.089,159.699
C09492=1017.037,-126.223,-97.583,165.027,55.083,159.698
C09493=1017.042,-125.973,-97.590,165.030,55.077,159.698
C09494=1017.047,-125.723,-97.597,165.034,55.073,159.698
C09495=1017.051,-125.473,-97.604,165.036,55.067,159.698
C09496=1017.057,-125.223,-97.611,165.039,55.061,159.697
C09497=1017.061,-124.973,-97.619,165.042,55.056,159.697
C09498=1017.067,-124.723,-97.626,165.045,55.051,159.697
C09499=1017.072,-124.473,-97.633,165.048,55.045,159.697
C09500=1017.076,-124.223,-97.641,165.051,55.039,159.696
C09501=1017.082,-123.974,-97.648,165.054,55.034,159.696
C09502=1017.087,-123.723,-97.655,165.057,55.029,159.696
C09503=1017.091,-123.474,-97.664,165.060,55.023,159.695
C09504=1017.097,-123.224,-97.671,165.063,55.018,159.695
C09505=1017.101,-122.975,-97.678,165.066,55.013,159.695
C09506=1017.106,-122.724,-97.686,165.069,55.007,159.695
C09507=1017.111,-122.475,-97.693,165.072,55.002,159.694
C09508=1017.116,-122.225,-97.701,165.075,54.996,159.694
C09509=1017.121,-121.975,-97.707,165.078,54.991,159.694
C09510=1017.126,-121.725,-97.715,165.081,54.985,159.694
C09511=1017.131,-121.475,-97.723,165.084,54.980,159.693
C09512=1017.136,-121.225,-97.730,165.087,54.974,159.693
C09513=1017.141,-120.976,-97.738,165.090,54.969,159.693
C09514=1017.146,-120.726,-97.746,165.093,54.964,159.693
C09515=1017.151,-120.476,-97.753,165.096,54.958,159.692
C09516=1017.156,-120.226,-97.760,165.098,54.952,159.692
C09517=1017.161,-119.976,-97.768,165.102,54.948,159.692
C09518=1017.166,-119.727,-97.776,165.105,54.942,159.691
C09519=1017.171,-119.477,-97.783,165.107,54.936,159.691
C09520=1017.176,-119.227,-97.791,165.110,54.931,159.691
C09521=1017.181,-118.977,-97.798,165.114,54.926,159.691
C09522=1017.186,-118.727,-97.806,165.116,54.920,159.690
C09523=1017.191,-118.478,-97.814,165.119,54.915,159.690
C09524=1017.197,-118.194,-97.822,165.123,54.909,159.690
C09525=1017.203,-117.911,-97.831,165.127,54.902,159.689
C09526=1017.208,-117.628,-97.839,165.130,54.896,159.689
C09527=1017.214,-117.345,-97.849,165.133,54.889,159.689
C09528=1017.219,-117.095,-97.856,165.136,54.885,159.689
C09529=1017.224,-116.845,-97.863,165.139,54.879,159.688
C09530=1017.229,-116.595,-97.872,165.142,54.873,159.688
C09531=1017.234,-116.345,-97.880,165.145,54.868,159.688
C09532=1017.239,-116.096,-97.886,165.148,54.863,159.687
C09533=1017.244,-115.846,-97.895,165.151,54.857,159.687
C09534=1017.249,-115.596,-97.903,165.154,54.852,159.687
C09535=1017.254,-115.346,-97.910,165.158,54.846,159.687
C09536=1017.260,-115.097,-97.918,165.160,54.840,159.686
C09537=1017.265,-114.846,-97.926,165.164,54.835,159.686
C09538=1017.270,-114.596,-97.934,165.167,54.830,159.686
C09539=1017.274,-114.347,-97.942,165.169,54.824,159.686
C09540=1017.279,-114.097,-97.949,165.172,54.818,159.685
C09541=1017.284,-113.847,-97.958,165.176,54.813,159.685
C09542=1017.290,-113.598,-97.965,165.178,54.808,159.685
C09543=1017.295,-113.348,-97.973,165.181,54.802,159.684
C09544=1017.300,-113.098,-97.981,165.184,54.797,159.684
C09545=1017.305,-112.848,-97.989,165.188,54.792,159.684
C09546=1017.309,-112.598,-97.997,165.190,54.786,159.684
C09547=1017.315,-112.348,-98.005,165.193,54.781,159.683
C09548=1017.320,-112.098,-98.013,165.196,54.775,159.683
C09549=1017.325,-111.848,-98.022,165.199,54.769,159.683
C09550=1017.330,-111.599,-98.028,165.202,54.765,159.683
C09551=1017.335,-111.349,-98.037,165.205,54.759,159.682
C09552=1017.340,-111.099,-98.045,165.208,54.753,159.682
C09553=1017.345,-110.849,-98.053,165.211,54.748,159.681
C09554=1017.350,-110.599,-98.061,165.214,54.742,159.681
C09555=1017.355,-110.350,-98.069,165.217,54.737,159.681
C09556=1017.360,-110.100,-98.077,165.220,54.732,159.681
C09557=1017.365,-109.850,-98.085,165.223,54.726,159.680
C09558=1017.371,-109.600,-98.094,165.226,54.720,159.680
C09559=1017.376,-109.350,-98.101,165.228,54.715,159.680
C09560=1017.381,-109.101,-98.109,165.232,54.710,159.680
C09561=1017.386,-108.851,-98.117,165.235,54.704,159.679
C09562=1017.391,-108.601,-98.125,165.239,54.698,159.679
C09563=1017.396,-108.351,-98.134,165.241,54.693,159.679
C09564=1017.401,-108.101,-98.142,165.244,54.687,159.678
C09565=1017.407,-107.851,-98.150,165.247,54.682,159.678
C09566=1017.412,-107.602,-98.159,165.250,54.677,159.678
C09567=1017.416,-107.352,-98.166,165.253,54.671,159.678
C09568=1017.421,-107.102,-98.174,165.256,54.666,159.677
C09569=1017.427,-106.853,-98.183,165.259,54.660,159.677
C09570=1017.432,-106.603,-98.191,165.262,54.654,159.677
C09571=1017.437,-106.353,-98.199,165.265,54.650,159.676
C09572=1017.442,-106.103,-98.208,165.268,54.644,159.676
C09573=1017.448,-105.853,-98.216,165.271,54.638,159.676
C09574=1017.453,-105.603,-98.225,165.274,54.633,159.675
C09575=1017.458,-105.353,-98.232,165.277,54.628,159.675
C09576=1017.463,-105.103,-98.241,165.280,54.622,159.675
C09577=1017.468,-104.854,-98.249,165.283,54.617,159.675
C09578=1017.473,-104.605,-98.257,165.286,54.611,159.674
C09579=1017.477,-104.355,-98.267,165.289,54.606,159.674
C09580=1017.482,-104.104,-98.274,165.292,54.601,159.674
C09581=1017.488,-103.855,-98.283,165.295,54.595,159.673
C09582=1017.493,-103.605,-98.291,165.298,54.590,159.673
C09583=1017.498,-103.355,-98.300,165.301,54.584,159.673
C09584=1017.503,-103.105,-98.308,165.304,54.579,159.673
C09585=1017.509,-102.856,-98.317,165.307,54.574,159.672
C09586=1017.514,-102.606,-98.325,165.310,54.568,159.672
C09587=1017.519,-102.356,-98.334,165.313,54.562,159.672
C09588=1017.525,-102.073,-98.343,165.316,54.557,159.671
C09589=1017.531,-101.790,-98.353,165.320,54.550,159.671
C09590=1017.537,-101.506,-98.363,165.324,54.544,159.671
C09591=1017.542,-101.224,-98.373,165.326,54.538,159.670
C09592=1017.547,-100.974,-98.381,165.329,54.532,159.670
C09593=1017.552,-100.723,-98.389,165.332,54.527,159.670
C09594=1017.557,-100.474,-98.397,165.336,54.521,159.670
C09595=1017.563,-100.224,-98.406,165.339,54.516,159.669
C09596=1017.568,-99.974,-98.414,165.342,54.510,159.669
C09597=1017.573,-99.725,-98.423,165.345,54.504,159.669
C09598=1017.578,-99.475,-98.431,165.348,54.499,159.668
C09599=1017.584,-99.225,-98.440,165.351,54.493,159.668
C09600=1017.588,-98.975,-98.449,165.354,54.488,159.668
C09601=1017.594,-98.725,-98.458,165.357,54.483,159.667
C09602=1017.599,-98.475,-98.466,165.360,54.477,159.667
C09603=1017.605,-98.225,-98.475,165.363,54.472,159.667
C09604=1017.610,-97.976,-98.483,165.366,54.466,159.666
C09605=1017.615,-97.726,-98.492,165.369,54.461,159.666
C09606=1017.620,-97.476,-98.501,165.371,54.455,159.666
C09607=1017.625,-97.227,-98.510,165.375,54.450,159.666
C09608=1017.630,-96.977,-98.519,165.378,54.445,159.665
C09609=1017.635,-96.727,-98.527,165.380,54.439,159.665
C09610=1017.640,-96.477,-98.536,165.384,54.434,159.665
C09611=1017.646,-96.227,-98.546,165.387,54.429,159.664
C09612=1017.651,-95.977,-98.555,165.390,54.423,159.664
C09613=1017.656,-95.727,-98.564,165.393,54.418,159.664
C09614=1017.661,-95.478,-98.572,165.396,54.413,159.664
C09615=1017.666,-95.228,-98.581,165.399,54.407,159.663
C09616=1017.671,-94.979,-98.590,165.402,54.402,159.663
C09617=1017.676,-94.729,-98.599,165.405,54.397,159.663
C09618=1017.681,-94.479,-98.608,165.408,54.391,159.662
C09619=1017.687,-94.228,-98.617,165.411,54.386,159.662
C09620=1017.692,-93.979,-98.626,165.414,54.380,159.662
C09621=1017.697,-93.729,-98.635,165.417,54.375,159.662
C09622=1017.702,-93.480,-98.644,165.420,54.370,159.661
C09623=1017.707,-93.230,-98.653,165.423,54.364,159.661
C09624=1017.712,-92.980,-98.662,165.426,54.359,159.661
C09625=1017.718,-92.730,-98.671,165.429,54.353,159.660
C09626=1017.723,-92.481,-98.681,165.432,54.348,159.660
C09627=1017.728,-92.231,-98.689,165.435,54.343,159.660
C09628=1017.733,-91.981,-98.698,165.438,54.337,159.659
C09629=1017.738,-91.732,-98.707,165.441,54.332,159.659
C09630=1017.744,-91.481,-98.716,165.443,54.326,159.659
C09631=1017.748,-91.231,-98.725,165.447,54.321,159.659
C09632=1017.754,-90.982,-98.734,165.450,54.316,159.658
C09633=1017.759,-90.732,-98.744,165.453,54.310,159.658
C09634=1017.764,-90.482,-98.752,165.456,54.305,159.658
C09635=1017.769,-90.232,-98.762,165.458,54.299,159.657
C09636=1017.775,-89.983,-98.771,165.462,54.294,159.657
C09637=1017.780,-89.734,-98.780,165.465,54.289,159.657
C09638=1017.785,-89.483,-98.789,165.468,54.283,159.656
C09639=1017.791,-89.234,-98.798,165.471,54.277,159.656
C09640=1017.795,-88.984,-98.808,165.474,54.272,159.656
C09641=1017.801,-88.734,-98.816,165.477,54.266,159.655
C09642=1017.807,-88.484,-98.826,165.480,54.261,159.655
C09643=1017.811,-88.234,-98.835,165.484,54.256,159.655
C09644=1017.817,-87.985,-98.844,165.486,54.250,159.655
C09645=1017.822,-87.734,-98.853,165.489,54.245,159.654
C09646=1017.828,-87.485,-98.863,165.492,54.239,159.654
C09647=1017.832,-87.235,-98.872,165.495,54.234,159.654
C09648=1017.838,-86.986,-98.881,165.498,54.228,159.653
C09649=1017.844,-86.736,-98.890,165.501,54.223,159.653
C09650=1017.848,-86.486,-98.899,165.504,54.217,159.653
C09651=1017.854,-86.237,-98.908,165.507,54.211,159.652
C09652=1017.860,-85.955,-98.919,165.511,54.206,159.652
C09653=1017.866,-85.675,-98.929,165.514,54.199,159.652
C09654=1017.872,-85.393,-98.940,165.517,54.193,159.651
C09655=1017.878,-85.112,-98.950,165.521,54.187,159.651
C09656=1017.883,-84.862,-98.960,165.523,54.181,159.650
C09657=1017.888,-84.613,-98.969,165.526,54.176,159.650
C09658=1017.893,-84.363,-98.978,165.529,54.170,159.650
C09659=1017.899,-84.113,-98.987,165.532,54.165,159.649
C09660=1017.904,-83.863,-98.997,165.536,54.159,159.649
C09661=1017.910,-83.613,-99.006,165.539,54.153,159.649
C09662=1017.915,-83.364,-99.015,165.542,54.148,159.648
C09663=1017.920,-83.114,-99.025,165.545,54.142,159.648
C09664=1017.926,-82.864,-99.034,165.548,54.137,159.648
C09665=1017.931,-82.615,-99.043,165.551,54.131,159.647
C09666=1017.937,-82.365,-99.053,165.554,54.125,159.647
C09667=1017.942,-82.115,-99.062,165.556,54.120,159.647
C09668=1017.947,-81.866,-99.071,165.559,54.114,159.646
C09669=1017.952,-81.615,-99.081,165.562,54.109,159.646
C09670=1017.958,-81.366,-99.090,165.566,54.103,159.646
C09671=1017.963,-81.116,-99.100,165.569,54.097,159.645
C09672=1017.969,-80.867,-99.109,165.572,54.092,159.645
C09673=1017.975,-80.616,-99.118,165.575,54.086,159.645
C09674=1017.980,-80.367,-99.128,165.578,54.081,159.644
C09675=1017.985,-80.117,-99.138,165.581,54.075,159.644
C09676=1017.990,-79.867,-99.147,165.584,54.071,159.644
C09677=1017.996,-79.617,-99.157,165.587,54.065,159.643
C09678=1018.001,-79.368,-99.167,165.590,54.060,159.643
C09679=1018.007,-79.118,-99.176,165.593,54.054,159.643
C09680=1018.012,-78.868,-99.186,165.596,54.048,159.642
C09681=1018.017,-78.618,-99.196,165.599,54.043,159.642
C09682=1018.022,-78.369,-99.206,165.602,54.038,159.642
C09683=1018.028,-78.119,-99.215,165.605,54.033,159.642
C09684=1018.033,-77.869,-99.225,165.608,54.027,159.641
C09685=1018.038,-77.619,-99.235,165.611,54.022,159.641
C09686=1018.044,-77.370,-99.244,165.614,54.016,159.640
C09687=1018.049,-77.120,-99.254,165.617,54.011,159.640
C09688=1018.054,-76.870,-99.264,165.620,54.005,159.640
C09689=1018.059,-76.620,-99.274,165.622,54.000,159.639
C09690=1018.065,-76.371,-99.283,165.625,53.994,159.639
C09691=1018.070,-76.121,-99.293,165.629,53.989,159.639
C09692=1018.075,-75.872,-99.303,165.632,53.984,159.638
C09693=1018.081,-75.621,-99.313,165.635,53.978,159.638
C09694=1018.087,-75.372,-99.323,165.638,53.973,159.638
C09695=1018.092,-75.122,-99.333,165.642,53.967,159.638
C09696=1018.097,-74.872,-99.343,165.644,53.961,159.637
C09697=1018.103,-74.623,-99.352,165.647,53.956,159.637
C09698=1018.108,-74.373,-99.362,165.650,53.950,159.636
C09699=1018.113,-74.123,-99.372,165.653,53.946,159.636
C09700=1018.118,-73.873,-99.382,165.656,53.940,159.636
C09701=1018.124,-73.623,-99.392,165.658,53.935,159.635
C09702=1018.128,-73.374,-99.403,165.661,53.929,159.635
C09703=1018.134,-73.124,-99.414,165.665,53.925,159.635
C09704=1018.139,-72.874,-99.424,165.668,53.919,159.635
C09705=1018.144,-72.625,-99.434,165.671,53.914,159.634
C09706=1018.149,-72.374,-99.444,165.674,53.908,159.634
C09707=1018.154,-72.125,-99.454,165.677,53.903,159.634
C09708=1018.159,-71.875,-99.464,165.680,53.898,159.633
C09709=1018.165,-71.625,-99.475,165.683,53.892,159.633
C09710=1018.170,-71.376,-99.484,165.686,53.887,159.633
C09711=1018.175,-71.126,-99.494,165.689,53.882,159.632
C09712=1018.181,-70.876,-99.505,165.692,53.877,159.632
C09713=1018.186,-70.627,-99.515,165.694,53.871,159.632
C09714=1018.192,-70.377,-99.525,165.697,53.866,159.631
C09715=1018.197,-70.127,-99.535,165.700,53.860,159.631
C09716=1018.202,-69.848,-99.547,165.704,53.855,159.631
C09717=1018.209,-69.569,-99.559,165.707,53.849,159.630
C09718=1018.214,-69.290,-99.570,165.710,53.842,159.630
C09719=1018.221,-69.011,-99.581,165.713,53.837,159.629
C09720=1018.226,-68.761,-99.591,165.716,53.831,159.629
C09721=1018.231,-68.511,-99.602,165.719,53.826,159.629
C09722=1018.237,-68.262,-99.612,165.722,53.821,159.629
C09723=1018.242,-68.012,-99.622,165.725,53.816,159.628
C09724=1018.247,-67.762,-99.632,165.728,53.810,159.628
C09725=1018.252,-67.512,-99.644,165.731,53.805,159.628
C09726=1018.257,-67.263,-99.654,165.734,53.799,159.627
C09727=1018.263,-67.013,-99.664,165.737,53.794,159.627
C09728=1018.268,-66.763,-99.675,165.740,53.788,159.626
C09729=1018.274,-66.513,-99.685,165.743,53.783,159.626
C09730=1018.279,-66.264,-99.695,165.746,53.778,159.626
C09731=1018.284,-66.014,-99.706,165.749,53.773,159.626
C09732=1018.291,-65.686,-99.720,165.753,53.765,159.625
C09733=1018.299,-65.357,-99.733,165.757,53.758,159.625
C09734=1018.306,-65.028,-99.747,165.761,53.751,159.624
C09735=1018.313,-64.699,-99.761,165.765,53.744,159.624
C09736=1018.318,-64.450,-99.771,165.767,53.738,159.623
C09737=1018.323,-64.200,-99.781,165.770,53.733,159.623
C09738=1018.329,-63.950,-99.791,165.773,53.728,159.623
C09739=1018.334,-63.701,-99.802,165.776,53.722,159.622
C09740=1018.340,-63.451,-99.812,165.779,53.717,159.622
C09741=1018.346,-63.201,-99.823,165.782,53.711,159.621
C09742=1018.350,-62.952,-99.833,165.786,53.706,159.621
C09743=1018.356,-62.702,-99.844,165.789,53.701,159.621
C09744=1018.362,-62.452,-99.854,165.791,53.695,159.621
C09745=1018.367,-62.203,-99.865,165.794,53.690,159.620
C09746=1018.373,-61.953,-99.875,165.797,53.684,159.620
C09747=1018.379,-61.703,-99.886,165.800,53.679,159.619
C09748=1018.384,-61.453,-99.896,165.803,53.673,159.619
C09749=1018.389,-61.204,-99.907,165.806,53.668,159.619
C09750=1018.394,-60.954,-99.918,165.809,53.662,159.618
C09751=1018.400,-60.704,-99.928,165.812,53.657,159.618
C09752=1018.405,-60.454,-99.939,165.815,53.652,159.618
C09753=1018.411,-60.205,-99.949,165.818,53.646,159.617
C09754=1018.416,-59.955,-99.960,165.821,53.641,159.617
C09755=1018.422,-59.705,-99.970,165.824,53.635,159.616
C09756=1018.428,-59.456,-99.981,165.827,53.630,159.616
C09757=1018.433,-59.205,-99.992,165.830,53.624,159.616
C09758=1018.439,-58.956,-100.002,165.833,53.619,159.615
C09759=1018.444,-58.707,-100.013,165.836,53.613,159.615
C09760=1018.449,-58.457,-100.023,165.839,53.608,159.615
C09761=1018.455,-58.208,-100.034,165.842,53.602,159.614
C09762=1018.460,-57.957,-100.045,165.844,53.597,159.614
C09763=1018.466,-57.708,-100.056,165.848,53.590,159.613
C09764=1018.471,-57.458,-100.066,165.851,53.585,159.613
C09765=1018.477,-57.208,-100.077,165.854,53.579,159.613
C09766=1018.482,-56.959,-100.088,165.857,53.574,159.612
C09767=1018.488,-56.709,-100.098,165.860,53.568,159.612
C09768=1018.494,-56.459,-100.109,165.863,53.563,159.612
C09769=1018.499,-56.209,-100.119,165.866,53.557,159.611
C09770=1018.505,-55.960,-100.130,165.869,53.552,159.611
C09771=1018.511,-55.710,-100.140,165.872,53.547,159.610
C09772=1018.516,-55.460,-100.151,165.875,53.541,159.610
C09773=1018.521,-55.211,-100.163,165.878,53.536,159.610
C09774=1018.527,-54.961,-100.174,165.881,53.530,159.609
C09775=1018.532,-54.711,-100.184,165.883,53.524,159.609
C09776=1018.537,-54.487,-100.194,165.886,53.519,159.609
C09777=1018.544,-54.263,-100.203,165.888,53.514,159.608
C09778=1018.548,-54.038,-100.213,165.892,53.509,159.608
///RCONF 1,0,0,0,0,0,0,0,0,0,0,0,0,0,0,0,0,0,0,0,0,0,0,0
C09779=1018.553,-53.814,-100.222,165.894,53.504,159.607
C09780=1018.558,-53.590,-100.232,165.897,53.499,159.607
C09781=1018.563,-53.364,-100.242,165.899,53.495,159.607
C09782=1018.568,-53.140,-100.252,165.902,53.489,159.606
C09783=1018.573,-52.916,-100.262,165.904,53.484,159.606
C09784=1018.579,-52.667,-100.272,165.907,53.479,159.605
C09785=1018.584,-52.417,-100.283,165.910,53.473,159.605
C09786=1018.590,-52.167,-100.294,165.914,53.467,159.605
C09787=1018.596,-51.917,-100.305,165.917,53.462,159.604
C09788=1018.602,-51.668,-100.316,165.920,53.456,159.604
C09789=1018.608,-51.418,-100.327,165.922,53.450,159.603
C09790=1018.612,-51.168,-100.337,165.925,53.445,159.603
C09791=1018.618,-50.918,-100.348,165.928,53.439,159.603
C09792=1018.624,-50.669,-100.359,165.931,53.434,159.602
C09793=1018.629,-50.419,-100.371,165.934,53.428,159.602
C09794=1018.635,-50.169,-100.381,165.936,53.423,159.601
C09795=1018.640,-49.920,-100.393,165.939,53.419,159.601
C09796=1018.645,-49.670,-100.404,165.942,53.413,159.601
C09797=1018.651,-49.420,-100.416,165.945,53.408,159.600
C09798=1018.657,-49.171,-100.427,165.948,53.402,159.600
C09799=1018.662,-48.921,-100.439,165.951,53.397,159.600
C09800=1018.668,-48.671,-100.450,165.954,53.391,159.599
C09801=1018.673,-48.422,-100.461,165.957,53.386,159.599
C09802=1018.678,-48.172,-100.472,165.960,53.380,159.599
C09803=1018.683,-47.922,-100.483,165.963,53.375,159.598
C09804=1018.689,-47.673,-100.494,165.966,53.370,159.598
C09805=1018.695,-47.422,-100.506,165.969,53.364,159.597
C09806=1018.700,-47.173,-100.517,165.971,53.359,159.597
C09807=1018.705,-46.923,-100.528,165.974,53.354,159.597
C09808=1018.712,-46.674,-100.540,165.977,53.348,159.596
C09809=1018.717,-46.424,-100.551,165.980,53.343,159.596
C09810=1018.722,-46.175,-100.562,165.983,53.337,159.595
C09811=1018.728,-45.924,-100.574,165.986,53.332,159.595
C09812=1018.734,-45.675,-100.585,165.989,53.326,159.595
C09813=1018.739,-45.425,-100.597,165.992,53.321,159.594
C09814=1018.745,-45.176,-100.608,165.995,53.316,159.594
C09815=1018.750,-44.926,-100.620,165.998,53.310,159.593
C09816=1018.755,-44.676,-100.631,166.001,53.305,159.593
C09817=1018.761,-44.426,-100.642,166.004,53.299,159.593
C09818=1018.766,-44.177,-100.654,166.007,53.294,159.592
C09819=1018.772,-43.928,-100.665,166.010,53.288,159.592
C09820=1018.777,-43.678,-100.677,166.013,53.283,159.592
C09821=1018.783,-43.428,-100.688,166.015,53.278,159.591
C09822=1018.788,-43.178,-100.700,166.018,53.272,159.591
C09823=1018.794,-42.929,-100.711,166.021,53.267,159.590
C09824=1018.799,-42.679,-100.723,166.024,53.262,159.590
C09825=1018.806,-42.429,-100.734,166.027,53.256,159.590
C09826=1018.811,-42.179,-100.745,166.030,53.251,159.589
C09827=1018.817,-41.931,-100.757,166.033,53.245,159.589
C09828=1018.822,-41.680,-100.769,166.036,53.240,159.588
C09829=1018.828,-41.431,-100.780,166.038,53.234,159.588
C09830=1018.833,-41.181,-100.792,166.041,53.228,159.587
C09831=1018.839,-40.932,-100.803,166.044,53.223,159.587
C09832=1018.845,-40.681,-100.815,166.047,53.217,159.587
C09833=1018.850,-40.432,-100.826,166.050,53.212,159.586
C09834=1018.856,-40.183,-100.838,166.053,53.207,159.586
C09835=1018.861,-39.932,-100.849,166.056,53.201,159.585
C09836=1018.867,-39.683,-100.860,166.059,53.196,159.585
C09837=1018.873,-39.433,-100.873,166.062,53.190,159.585
C09838=1018.879,-39.183,-100.884,166.065,53.185,159.584
C09839=1018.884,-38.934,-100.896,166.068,53.180,159.584
C09840=1018.889,-38.684,-100.907,166.070,53.174,159.583
C09841=1018.895,-38.434,-100.920,166.073,53.169,159.583
C09842=1018.900,-38.185,-100.931,166.076,53.164,159.583
C09843=1018.906,-37.936,-100.943,166.079,53.158,159.582
C09844=1018.912,-37.658,-100.956,166.081,53.152,159.582
C09845=1018.919,-37.380,-100.970,166.085,53.146,159.581
C09846=1018.925,-37.102,-100.983,166.088,53.140,159.581
C09847=1018.931,-36.825,-100.996,166.092,53.134,159.581
C09848=1018.936,-36.575,-101.008,166.095,53.129,159.580
C09849=1018.942,-36.325,-101.020,166.097,53.124,159.580
C09850=1018.947,-36.076,-101.032,166.100,53.118,159.579
C09851=1018.952,-35.826,-101.043,166.103,53.113,159.579
C09852=1018.959,-35.576,-101.055,166.106,53.108,159.578
C09853=1018.964,-35.326,-101.067,166.108,53.102,159.578
C09854=1018.970,-35.077,-101.079,166.111,53.096,159.577
C09855=1018.975,-34.827,-101.092,166.114,53.091,159.577
C09856=1018.980,-34.578,-101.103,166.117,53.085,159.577
C09857=1018.986,-34.328,-101.115,166.119,53.080,159.576
C09858=1018.991,-34.078,-101.126,166.122,53.075,159.576
C09859=1018.997,-33.828,-101.139,166.125,53.069,159.575
C09860=1019.003,-33.579,-101.151,166.128,53.064,159.575
C09861=1019.008,-33.329,-101.163,166.131,53.059,159.575
C09862=1019.014,-33.079,-101.175,166.134,53.053,159.574
C09863=1019.020,-32.831,-101.187,166.137,53.048,159.574
C09864=1019.025,-32.580,-101.199,166.140,53.042,159.573
C09865=1019.031,-32.331,-101.211,166.143,53.037,159.573
C09866=1019.036,-32.081,-101.223,166.145,53.032,159.573
C09867=1019.041,-31.831,-101.235,166.148,53.027,159.572
C09868=1019.048,-31.582,-101.247,166.151,53.020,159.572
C09869=1019.053,-31.333,-101.259,166.154,53.015,159.571
C09870=1019.059,-31.082,-101.271,166.157,53.010,159.571
C09871=1019.064,-30.833,-101.283,166.160,53.004,159.570
C09872=1019.070,-30.584,-101.295,166.163,52.999,159.570
C09873=1019.076,-30.334,-101.308,166.166,52.993,159.570
C09874=1019.081,-30.084,-101.319,166.169,52.988,159.569
C09875=1019.087,-29.834,-101.331,166.172,52.983,159.569
C09876=1019.092,-29.585,-101.343,166.174,52.977,159.568
C09877=1019.098,-29.335,-101.355,166.176,52.972,159.568
C09878=1019.104,-29.085,-101.368,166.179,52.966,159.567
C09879=1019.109,-28.836,-101.380,166.182,52.961,159.567
C09880=1019.116,-28.586,-101.392,166.185,52.955,159.567
C09881=1019.121,-28.337,-101.404,166.188,52.950,159.566
C09882=1019.127,-28.086,-101.416,166.191,52.944,159.566
C09883=1019.132,-27.837,-101.428,166.194,52.938,159.565
C09884=1019.138,-27.587,-101.441,166.197,52.933,159.565
C09885=1019.143,-27.338,-101.453,166.200,52.928,159.564
C09886=1019.149,-27.088,-101.465,166.202,52.923,159.564
C09887=1019.155,-26.838,-101.478,166.205,52.917,159.563
C09888=1019.161,-26.589,-101.490,166.208,52.912,159.563
C09889=1019.166,-26.339,-101.503,166.211,52.906,159.563
C09890=1019.172,-26.090,-101.515,166.214,52.901,159.562
C09891=1019.177,-25.839,-101.527,166.217,52.896,159.562
C09892=1019.182,-25.590,-101.540,166.219,52.891,159.561
C09893=1019.188,-25.340,-101.552,166.222,52.885,159.561
C09894=1019.194,-25.090,-101.565,166.225,52.880,159.561
C09895=1019.199,-24.841,-101.577,166.228,52.875,159.560
C09896=1019.205,-24.591,-101.589,166.231,52.869,159.560
C09897=1019.210,-24.342,-101.602,166.234,52.864,159.559
C09898=1019.216,-24.092,-101.614,166.236,52.859,159.559
C09899=1019.221,-23.843,-101.628,166.239,52.853,159.558
C09900=1019.227,-23.593,-101.640,166.242,52.847,159.558
C09901=1019.233,-23.344,-101.653,166.245,52.842,159.557
C09902=1019.238,-23.094,-101.665,166.248,52.836,159.557
C09903=1019.244,-22.845,-101.678,166.251,52.831,159.557
C09904=1019.250,-22.595,-101.690,166.253,52.826,159.556
C09905=1019.255,-22.345,-101.702,166.256,52.821,159.556
C09906=1019.261,-22.096,-101.715,166.259,52.815,159.555
C09907=1019.267,-21.846,-101.727,166.262,52.810,159.555
C09908=1019.273,-21.567,-101.741,166.264,52.804,159.554
C09909=1019.279,-21.288,-101.755,166.268,52.797,159.554
C09910=1019.286,-21.011,-101.770,166.271,52.791,159.553
C09911=1019.292,-20.732,-101.784,166.275,52.786,159.553
C09912=1019.298,-20.482,-101.796,166.277,52.781,159.552
C09913=1019.303,-20.232,-101.809,166.279,52.774,159.552
C09914=1019.309,-19.983,-101.821,166.282,52.769,159.551
C09915=1019.314,-19.733,-101.834,166.285,52.764,159.551
C09916=1019.320,-19.483,-101.847,166.288,52.758,159.551
C09917=1019.325,-19.234,-101.860,166.291,52.753,159.550
C09918=1019.331,-18.985,-101.872,166.293,52.748,159.550
C09919=1019.337,-18.735,-101.885,166.296,52.742,159.549
C09920=1019.343,-18.485,-101.897,166.299,52.737,159.549
C09921=1019.348,-18.236,-101.909,166.302,52.731,159.548
C09922=1019.354,-17.986,-101.922,166.305,52.726,159.548
C09923=1019.360,-17.736,-101.936,166.308,52.720,159.547
C09924=1019.365,-17.487,-101.948,166.311,52.714,159.547
C09925=1019.371,-17.237,-101.961,166.314,52.709,159.547
C09926=1019.377,-16.987,-101.973,166.316,52.704,159.546
C09927=1019.383,-16.738,-101.986,166.319,52.699,159.546
C09928=1019.388,-16.489,-101.999,166.321,52.693,159.545
C09929=1019.394,-16.239,-102.011,166.324,52.687,159.545
C09930=1019.400,-15.989,-102.024,166.327,52.682,159.544
C09931=1019.406,-15.739,-102.038,166.330,52.676,159.544
C09932=1019.411,-15.490,-102.050,166.332,52.671,159.543
C09933=1019.416,-15.240,-102.063,166.335,52.666,159.543
C09934=1019.422,-14.991,-102.076,166.338,52.660,159.542
C09935=1019.428,-14.741,-102.089,166.341,52.655,159.542
C09936=1019.433,-14.492,-102.102,166.344,52.649,159.541
C09937=1019.439,-14.242,-102.115,166.346,52.644,159.541
C09938=1019.444,-13.992,-102.128,166.349,52.639,159.540
C09939=1019.451,-13.743,-102.141,166.352,52.634,159.540
C09940=1019.456,-13.492,-102.154,166.355,52.628,159.540
C09941=1019.461,-13.244,-102.167,166.357,52.623,159.539
C09942=1019.467,-12.994,-102.180,166.360,52.618,159.539
C09943=1019.473,-12.744,-102.194,166.363,52.612,159.538
C09944=1019.479,-12.495,-102.206,166.366,52.606,159.538
C09945=1019.484,-12.244,-102.219,166.369,52.601,159.537
C09946=1019.489,-11.996,-102.232,166.371,52.596,159.537
C09947=1019.495,-11.746,-102.245,166.374,52.591,159.536
C09948=1019.501,-11.496,-102.259,166.377,52.585,159.536
C09949=1019.507,-11.246,-102.271,166.380,52.579,159.535
C09950=1019.512,-10.997,-102.285,166.383,52.574,159.535
C09951=1019.518,-10.747,-102.298,166.385,52.569,159.534
C09952=1019.523,-10.498,-102.311,166.388,52.564,159.534
C09953=1019.529,-10.248,-102.324,166.391,52.558,159.534
C09954=1019.535,-9.999,-102.337,166.393,52.552,159.533
C09955=1019.540,-9.749,-102.350,166.396,52.547,159.533
C09956=1019.546,-9.500,-102.363,166.398,52.542,159.532
C09957=1019.552,-9.250,-102.377,166.401,52.537,159.532
C09958=1019.558,-9.000,-102.390,166.404,52.531,159.531
C09959=1019.563,-8.750,-102.404,166.407,52.525,159.531
C09960=1019.569,-8.501,-102.416,166.410,52.520,159.530
C09961=1019.575,-8.252,-102.429,166.413,52.515,159.530
C09962=1019.580,-8.002,-102.442,166.415,52.509,159.529
C09963=1019.586,-7.753,-102.456,166.418,52.503,159.529
C09964=1019.592,-7.503,-102.469,166.421,52.498,159.528
C09965=1019.598,-7.253,-102.482,166.424,52.493,159.528
C09966=1019.603,-7.004,-102.496,166.426,52.487,159.527
C09967=1019.609,-6.754,-102.508,166.430,52.481,159.527
C09968=1019.615,-6.504,-102.522,166.432,52.476,159.526
C09969=1019.621,-6.255,-102.536,166.434,52.470,159.526
C09970=1019.627,-6.005,-102.548,166.437,52.465,159.525
C09971=1019.632,-5.755,-102.562,166.440,52.460,159.525
C09972=1019.639,-5.476,-102.576,166.443,52.454,159.524
C09973=1019.645,-5.195,-102.591,166.447,52.447,159.524
C09974=1019.651,-4.915,-102.606,166.449,52.441,159.523
C09975=1019.658,-4.634,-102.621,166.453,52.435,159.523
C09976=1019.663,-4.385,-102.635,166.455,52.429,159.522
C09977=1019.669,-4.135,-102.648,166.457,52.424,159.522
C09978=1019.675,-3.885,-102.661,166.461,52.418,159.521
C09979=1019.680,-3.636,-102.675,166.464,52.413,159.521
C09980=1019.686,-3.386,-102.689,166.467,52.408,159.520
C09981=1019.692,-3.137,-102.702,166.469,52.403,159.520
C09982=1019.697,-2.887,-102.716,166.471,52.397,159.519
C09983=1019.703,-2.637,-102.729,166.474,52.391,159.519
C09984=1019.708,-2.388,-102.743,166.476,52.386,159.518
C09985=1019.714,-2.138,-102.757,166.479,52.381,159.518
C09986=1019.720,-1.889,-102.770,166.483,52.376,159.517
C09987=1019.725,-1.639,-102.784,166.486,52.370,159.517
C09988=1019.731,-1.390,-102.798,166.487,52.365,159.516
C09989=1019.736,-1.140,-102.812,166.490,52.359,159.516
C09990=1019.742,-0.891,-102.826,166.493,52.354,159.516
C09991=1019.748,-0.641,-102.839,166.496,52.349,159.515
C09992=1019.753,-0.392,-102.853,166.498,52.344,159.515
C09993=1019.759,-0.142,-102.867,166.501,52.338,159.514
C09994=1019.764,0.108,-102.880,166.504,52.333,159.514
C09995=1019.769,0.358,-102.894,166.507,52.327,159.513
C09996=1019.776,0.607,-102.907,166.509,52.322,159.513
//INST
///DATE 2021/06/17 10:59
///ATTR SC,RW,RJ
////FRAME ROBOT
///GROUP1 RB1
NOP
MOVL C00000 V=800.0 PL=0
MOVL C00001 V=800.0 PL=0
MOVL C00002 V=800.0 PL=0
MOVL C00003 V=800.0 PL=0
MOVL C00004 V=800.0 PL=0
MOVL C00005 V=800.0 PL=0
MOVL C00006 V=800.0 PL=0
MOVL C00007 V=800.0 PL=0
MOVL C00008 V=800.0 PL=0
MOVL C00009 V=800.0 PL=0
MOVL C00010 V=800.0 PL=0
MOVL C00011 V=800.0 PL=0
MOVL C00012 V=800.0 PL=0
MOVL C00013 V=800.0 PL=0
MOVL C00014 V=800.0 PL=0
MOVL C00015 V=800.0 PL=0
MOVL C00016 V=800.0 PL=0
MOVL C00017 V=800.0 PL=0
MOVL C00018 V=800.0 PL=0
MOVL C00019 V=800.0 PL=0
MOVL C00020 V=800.0 PL=0
MOVL C00021 V=800.0 PL=0
MOVL C00022 V=800.0 PL=0
MOVL C00023 V=800.0 PL=0
MOVL C00024 V=800.0 PL=0
MOVL C00025 V=800.0 PL=0
MOVL C00026 V=800.0 PL=0
MOVL C00027 V=800.0 PL=0
MOVL C00028 V=800.0 PL=0
MOVL C00029 V=800.0 PL=0
MOVL C00030 V=800.0 PL=0
MOVL C00031 V=800.0 PL=0
MOVL C00032 V=800.0 PL=0
MOVL C00033 V=800.0 PL=0
MOVL C00034 V=800.0 PL=0
MOVL C00035 V=800.0 PL=0
MOVL C00036 V=800.0 PL=0
MOVL C00037 V=800.0 PL=0
MOVL C00038 V=800.0 PL=0
MOVL C00039 V=800.0 PL=0
MOVL C00040 V=800.0 PL=0
MOVL C00041 V=800.0 PL=0
MOVL C00042 V=800.0 PL=0
MOVL C00043 V=800.0 PL=0
MOVL C00044 V=800.0 PL=0
MOVL C00045 V=800.0 PL=0
MOVL C00046 V=800.0 PL=0
MOVL C00047 V=800.0 PL=0
MOVL C00048 V=800.0 PL=0
MOVL C00049 V=800.0 PL=0
MOVL C00050 V=800.0 PL=0
MOVL C00051 V=800.0 PL=0
MOVL C00052 V=800.0 PL=0
MOVL C00053 V=800.0 PL=0
MOVL C00054 V=800.0 PL=0
MOVL C00055 V=800.0 PL=0
MOVL C00056 V=800.0 PL=0
MOVL C00057 V=800.0 PL=0
MOVL C00058 V=800.0 PL=0
MOVL C00059 V=800.0 PL=0
MOVL C00060 V=800.0 PL=0
MOVL C00061 V=800.0 PL=0
MOVL C00062 V=800.0 PL=0
MOVL C00063 V=800.0 PL=0
MOVL C00064 V=800.0 PL=0
MOVL C00065 V=800.0 PL=0
MOVL C00066 V=800.0 PL=0
MOVL C00067 V=800.0 PL=0
MOVL C00068 V=800.0 PL=0
MOVL C00069 V=800.0 PL=0
MOVL C00070 V=800.0 PL=0
MOVL C00071 V=800.0 PL=0
MOVL C00072 V=800.0 PL=0
MOVL C00073 V=800.0 PL=0
MOVL C00074 V=800.0 PL=0
MOVL C00075 V=800.0 PL=0
MOVL C00076 V=800.0 PL=0
MOVL C00077 V=800.0 PL=0
MOVL C00078 V=800.0 PL=0
MOVL C00079 V=800.0 PL=0
MOVL C00080 V=800.0 PL=0
MOVL C00081 V=800.0 PL=0
MOVL C00082 V=800.0 PL=0
MOVL C00083 V=800.0 PL=0
MOVL C00084 V=800.0 PL=0
MOVL C00085 V=800.0 PL=0
MOVL C00086 V=800.0 PL=0
MOVL C00087 V=800.0 PL=0
MOVL C00088 V=800.0 PL=0
MOVL C00089 V=800.0 PL=0
MOVL C00090 V=800.0 PL=0
MOVL C00091 V=800.0 PL=0
MOVL C00092 V=800.0 PL=0
MOVL C00093 V=800.0 PL=0
MOVL C00094 V=800.0 PL=0
MOVL C00095 V=800.0 PL=0
MOVL C00096 V=800.0 PL=0
MOVL C00097 V=800.0 PL=0
MOVL C00098 V=800.0 PL=0
MOVL C00099 V=800.0 PL=0
MOVL C00100 V=800.0 PL=0
MOVL C00101 V=800.0 PL=0
MOVL C00102 V=800.0 PL=0
MOVL C00103 V=800.0 PL=0
MOVL C00104 V=800.0 PL=0
MOVL C00105 V=800.0 PL=0
MOVL C00106 V=800.0 PL=0
MOVL C00107 V=800.0 PL=0
MOVL C00108 V=800.0 PL=0
MOVL C00109 V=800.0 PL=0
MOVL C00110 V=800.0 PL=0
MOVL C00111 V=800.0 PL=0
MOVL C00112 V=800.0 PL=0
MOVL C00113 V=800.0 PL=0
MOVL C00114 V=800.0 PL=0
MOVL C00115 V=800.0 PL=0
MOVL C00116 V=800.0 PL=0
MOVL C00117 V=800.0 PL=0
MOVL C00118 V=800.0 PL=0
MOVL C00119 V=800.0 PL=0
MOVL C00120 V=800.0 PL=0
MOVL C00121 V=800.0 PL=0
MOVL C00122 V=800.0 PL=0
MOVL C00123 V=800.0 PL=0
MOVL C00124 V=800.0 PL=0
MOVL C00125 V=800.0 PL=0
MOVL C00126 V=800.0 PL=0
MOVL C00127 V=800.0 PL=0
MOVL C00128 V=800.0 PL=0
MOVL C00129 V=800.0 PL=0
MOVL C00130 V=800.0 PL=0
MOVL C00131 V=800.0 PL=0
MOVL C00132 V=800.0 PL=0
MOVL C00133 V=800.0 PL=0
MOVL C00134 V=800.0 PL=0
MOVL C00135 V=800.0 PL=0
MOVL C00136 V=800.0 PL=0
MOVL C00137 V=800.0 PL=0
MOVL C00138 V=800.0 PL=0
MOVL C00139 V=800.0 PL=0
MOVL C00140 V=800.0 PL=0
MOVL C00141 V=800.0 PL=0
MOVL C00142 V=800.0 PL=0
MOVL C00143 V=800.0 PL=0
MOVL C00144 V=800.0 PL=0
MOVL C00145 V=800.0 PL=0
MOVL C00146 V=800.0 PL=0
MOVL C00147 V=800.0 PL=0
MOVL C00148 V=800.0 PL=0
MOVL C00149 V=800.0 PL=0
MOVL C00150 V=800.0 PL=0
MOVL C00151 V=800.0 PL=0
MOVL C00152 V=800.0 PL=0
MOVL C00153 V=800.0 PL=0
MOVL C00154 V=800.0 PL=0
MOVL C00155 V=800.0 PL=0
MOVL C00156 V=800.0 PL=0
MOVL C00157 V=800.0 PL=0
MOVL C00158 V=800.0 PL=0
MOVL C00159 V=800.0 PL=0
MOVL C00160 V=800.0 PL=0
MOVL C00161 V=800.0 PL=0
MOVL C00162 V=800.0 PL=0
MOVL C00163 V=800.0 PL=0
MOVL C00164 V=800.0 PL=0
MOVL C00165 V=800.0 PL=0
MOVL C00166 V=800.0 PL=0
MOVL C00167 V=800.0 PL=0
MOVL C00168 V=800.0 PL=0
MOVL C00169 V=800.0 PL=0
MOVL C00170 V=800.0 PL=0
MOVL C00171 V=800.0 PL=0
MOVL C00172 V=800.0 PL=0
MOVL C00173 V=800.0 PL=0
MOVL C00174 V=800.0 PL=0
MOVL C00175 V=800.0 PL=0
MOVL C00176 V=800.0 PL=0
MOVL C00177 V=800.0 PL=0
MOVL C00178 V=800.0 PL=0
MOVL C00179 V=800.0 PL=0
MOVL C00180 V=800.0 PL=0
MOVL C00181 V=800.0 PL=0
MOVL C00182 V=800.0 PL=0
MOVL C00183 V=800.0 PL=0
MOVL C00184 V=800.0 PL=0
MOVL C00185 V=800.0 PL=0
MOVL C00186 V=800.0 PL=0
MOVL C00187 V=800.0 PL=0
MOVL C00188 V=800.0 PL=0
MOVL C00189 V=800.0 PL=0
MOVL C00190 V=800.0 PL=0
MOVL C00191 V=800.0 PL=0
MOVL C00192 V=800.0 PL=0
MOVL C00193 V=800.0 PL=0
MOVL C00194 V=800.0 PL=0
MOVL C00195 V=800.0 PL=0
MOVL C00196 V=800.0 PL=0
MOVL C00197 V=800.0 PL=0
MOVL C00198 V=800.0 PL=0
MOVL C00199 V=800.0 PL=0
MOVL C00200 V=800.0 PL=0
MOVL C00201 V=800.0 PL=0
MOVL C00202 V=800.0 PL=0
MOVL C00203 V=800.0 PL=0
MOVL C00204 V=800.0 PL=0
MOVL C00205 V=800.0 PL=0
MOVL C00206 V=800.0 PL=0
MOVL C00207 V=800.0 PL=0
MOVL C00208 V=800.0 PL=0
MOVL C00209 V=800.0 PL=0
MOVL C00210 V=800.0 PL=0
MOVL C00211 V=800.0 PL=0
MOVL C00212 V=800.0 PL=0
MOVL C00213 V=800.0 PL=0
MOVL C00214 V=800.0 PL=0
MOVL C00215 V=800.0 PL=0
MOVL C00216 V=800.0 PL=0
MOVL C00217 V=800.0 PL=0
MOVL C00218 V=800.0 PL=0
MOVL C00219 V=800.0 PL=0
MOVL C00220 V=800.0 PL=0
MOVL C00221 V=800.0 PL=0
MOVL C00222 V=800.0 PL=0
MOVL C00223 V=800.0 PL=0
MOVL C00224 V=800.0 PL=0
MOVL C00225 V=800.0 PL=0
MOVL C00226 V=800.0 PL=0
MOVL C00227 V=800.0 PL=0
MOVL C00228 V=800.0 PL=0
MOVL C00229 V=800.0 PL=0
MOVL C00230 V=800.0 PL=0
MOVL C00231 V=800.0 PL=0
MOVL C00232 V=800.0 PL=0
MOVL C00233 V=800.0 PL=0
MOVL C00234 V=800.0 PL=0
MOVL C00235 V=800.0 PL=0
MOVL C00236 V=800.0 PL=0
MOVL C00237 V=800.0 PL=0
MOVL C00238 V=800.0 PL=0
MOVL C00239 V=800.0 PL=0
MOVL C00240 V=800.0 PL=0
MOVL C00241 V=800.0 PL=0
MOVL C00242 V=800.0 PL=0
MOVL C00243 V=800.0 PL=0
MOVL C00244 V=800.0 PL=0
MOVL C00245 V=800.0 PL=0
MOVL C00246 V=800.0 PL=0
MOVL C00247 V=800.0 PL=0
MOVL C00248 V=800.0 PL=0
MOVL C00249 V=800.0 PL=0
MOVL C00250 V=800.0 PL=0
MOVL C00251 V=800.0 PL=0
MOVL C00252 V=800.0 PL=0
MOVL C00253 V=800.0 PL=0
MOVL C00254 V=800.0 PL=0
MOVL C00255 V=800.0 PL=0
MOVL C00256 V=800.0 PL=0
MOVL C00257 V=800.0 PL=0
MOVL C00258 V=800.0 PL=0
MOVL C00259 V=800.0 PL=0
MOVL C00260 V=800.0 PL=0
MOVL C00261 V=800.0 PL=0
MOVL C00262 V=800.0 PL=0
MOVL C00263 V=800.0 PL=0
MOVL C00264 V=800.0 PL=0
MOVL C00265 V=800.0 PL=0
MOVL C00266 V=800.0 PL=0
MOVL C00267 V=800.0 PL=0
MOVL C00268 V=800.0 PL=0
MOVL C00269 V=800.0 PL=0
MOVL C00270 V=800.0 PL=0
MOVL C00271 V=800.0 PL=0
MOVL C00272 V=800.0 PL=0
MOVL C00273 V=800.0 PL=0
MOVL C00274 V=800.0 PL=0
MOVL C00275 V=800.0 PL=0
MOVL C00276 V=800.0 PL=0
MOVL C00277 V=800.0 PL=0
MOVL C00278 V=800.0 PL=0
MOVL C00279 V=800.0 PL=0
MOVL C00280 V=800.0 PL=0
MOVL C00281 V=800.0 PL=0
MOVL C00282 V=800.0 PL=0
MOVL C00283 V=800.0 PL=0
MOVL C00284 V=800.0 PL=0
MOVL C00285 V=800.0 PL=0
MOVL C00286 V=800.0 PL=0
MOVL C00287 V=800.0 PL=0
MOVL C00288 V=800.0 PL=0
MOVL C00289 V=800.0 PL=0
MOVL C00290 V=800.0 PL=0
MOVL C00291 V=800.0 PL=0
MOVL C00292 V=800.0 PL=0
MOVL C00293 V=800.0 PL=0
MOVL C00294 V=800.0 PL=0
MOVL C00295 V=800.0 PL=0
MOVL C00296 V=800.0 PL=0
MOVL C00297 V=800.0 PL=0
MOVL C00298 V=800.0 PL=0
MOVL C00299 V=800.0 PL=0
MOVL C00300 V=800.0 PL=0
MOVL C00301 V=800.0 PL=0
MOVL C00302 V=800.0 PL=0
MOVL C00303 V=800.0 PL=0
MOVL C00304 V=800.0 PL=0
MOVL C00305 V=800.0 PL=0
MOVL C00306 V=800.0 PL=0
MOVL C00307 V=800.0 PL=0
MOVL C00308 V=800.0 PL=0
MOVL C00309 V=800.0 PL=0
MOVL C00310 V=800.0 PL=0
MOVL C00311 V=800.0 PL=0
MOVL C00312 V=800.0 PL=0
MOVL C00313 V=800.0 PL=0
MOVL C00314 V=800.0 PL=0
MOVL C00315 V=800.0 PL=0
MOVL C00316 V=800.0 PL=0
MOVL C00317 V=800.0 PL=0
MOVL C00318 V=800.0 PL=0
MOVL C00319 V=800.0 PL=0
MOVL C00320 V=800.0 PL=0
MOVL C00321 V=800.0 PL=0
MOVL C00322 V=800.0 PL=0
MOVL C00323 V=800.0 PL=0
MOVL C00324 V=800.0 PL=0
MOVL C00325 V=800.0 PL=0
MOVL C00326 V=800.0 PL=0
MOVL C00327 V=800.0 PL=0
MOVL C00328 V=800.0 PL=0
MOVL C00329 V=800.0 PL=0
MOVL C00330 V=800.0 PL=0
MOVL C00331 V=800.0 PL=0
MOVL C00332 V=800.0 PL=0
MOVL C00333 V=800.0 PL=0
MOVL C00334 V=800.0 PL=0
MOVL C00335 V=800.0 PL=0
MOVL C00336 V=800.0 PL=0
MOVL C00337 V=800.0 PL=0
MOVL C00338 V=800.0 PL=0
MOVL C00339 V=800.0 PL=0
MOVL C00340 V=800.0 PL=0
MOVL C00341 V=800.0 PL=0
MOVL C00342 V=800.0 PL=0
MOVL C00343 V=800.0 PL=0
MOVL C00344 V=800.0 PL=0
MOVL C00345 V=800.0 PL=0
MOVL C00346 V=800.0 PL=0
MOVL C00347 V=800.0 PL=0
MOVL C00348 V=800.0 PL=0
MOVL C00349 V=800.0 PL=0
MOVL C00350 V=800.0 PL=0
MOVL C00351 V=800.0 PL=0
MOVL C00352 V=800.0 PL=0
MOVL C00353 V=800.0 PL=0
MOVL C00354 V=800.0 PL=0
MOVL C00355 V=800.0 PL=0
MOVL C00356 V=800.0 PL=0
MOVL C00357 V=800.0 PL=0
MOVL C00358 V=800.0 PL=0
MOVL C00359 V=800.0 PL=0
MOVL C00360 V=800.0 PL=0
MOVL C00361 V=800.0 PL=0
MOVL C00362 V=800.0 PL=0
MOVL C00363 V=800.0 PL=0
MOVL C00364 V=800.0 PL=0
MOVL C00365 V=800.0 PL=0
MOVL C00366 V=800.0 PL=0
MOVL C00367 V=800.0 PL=0
MOVL C00368 V=800.0 PL=0
MOVL C00369 V=800.0 PL=0
MOVL C00370 V=800.0 PL=0
MOVL C00371 V=800.0 PL=0
MOVL C00372 V=800.0 PL=0
MOVL C00373 V=800.0 PL=0
MOVL C00374 V=800.0 PL=0
MOVL C00375 V=800.0 PL=0
MOVL C00376 V=800.0 PL=0
MOVL C00377 V=800.0 PL=0
MOVL C00378 V=800.0 PL=0
MOVL C00379 V=800.0 PL=0
MOVL C00380 V=800.0 PL=0
MOVL C00381 V=800.0 PL=0
MOVL C00382 V=800.0 PL=0
MOVL C00383 V=800.0 PL=0
MOVL C00384 V=800.0 PL=0
MOVL C00385 V=800.0 PL=0
MOVL C00386 V=800.0 PL=0
MOVL C00387 V=800.0 PL=0
MOVL C00388 V=800.0 PL=0
MOVL C00389 V=800.0 PL=0
MOVL C00390 V=800.0 PL=0
MOVL C00391 V=800.0 PL=0
MOVL C00392 V=800.0 PL=0
MOVL C00393 V=800.0 PL=0
MOVL C00394 V=800.0 PL=0
MOVL C00395 V=800.0 PL=0
MOVL C00396 V=800.0 PL=0
MOVL C00397 V=800.0 PL=0
MOVL C00398 V=800.0 PL=0
MOVL C00399 V=800.0 PL=0
MOVL C00400 V=800.0 PL=0
MOVL C00401 V=800.0 PL=0
MOVL C00402 V=800.0 PL=0
MOVL C00403 V=800.0 PL=0
MOVL C00404 V=800.0 PL=0
MOVL C00405 V=800.0 PL=0
MOVL C00406 V=800.0 PL=0
MOVL C00407 V=800.0 PL=0
MOVL C00408 V=800.0 PL=0
MOVL C00409 V=800.0 PL=0
MOVL C00410 V=800.0 PL=0
MOVL C00411 V=800.0 PL=0
MOVL C00412 V=800.0 PL=0
MOVL C00413 V=800.0 PL=0
MOVL C00414 V=800.0 PL=0
MOVL C00415 V=800.0 PL=0
MOVL C00416 V=800.0 PL=0
MOVL C00417 V=800.0 PL=0
MOVL C00418 V=800.0 PL=0
MOVL C00419 V=800.0 PL=0
MOVL C00420 V=800.0 PL=0
MOVL C00421 V=800.0 PL=0
MOVL C00422 V=800.0 PL=0
MOVL C00423 V=800.0 PL=0
MOVL C00424 V=800.0 PL=0
MOVL C00425 V=800.0 PL=0
MOVL C00426 V=800.0 PL=0
MOVL C00427 V=800.0 PL=0
MOVL C00428 V=800.0 PL=0
MOVL C00429 V=800.0 PL=0
MOVL C00430 V=800.0 PL=0
MOVL C00431 V=800.0 PL=0
MOVL C00432 V=800.0 PL=0
MOVL C00433 V=800.0 PL=0
MOVL C00434 V=800.0 PL=0
MOVL C00435 V=800.0 PL=0
MOVL C00436 V=800.0 PL=0
MOVL C00437 V=800.0 PL=0
MOVL C00438 V=800.0 PL=0
MOVL C00439 V=800.0 PL=0
MOVL C00440 V=800.0 PL=0
MOVL C00441 V=800.0 PL=0
MOVL C00442 V=800.0 PL=0
MOVL C00443 V=800.0 PL=0
MOVL C00444 V=800.0 PL=0
MOVL C00445 V=800.0 PL=0
MOVL C00446 V=800.0 PL=0
MOVL C00447 V=800.0 PL=0
MOVL C00448 V=800.0 PL=0
MOVL C00449 V=800.0 PL=0
MOVL C00450 V=800.0 PL=0
MOVL C00451 V=800.0 PL=0
MOVL C00452 V=800.0 PL=0
MOVL C00453 V=800.0 PL=0
MOVL C00454 V=800.0 PL=0
MOVL C00455 V=800.0 PL=0
MOVL C00456 V=800.0 PL=0
MOVL C00457 V=800.0 PL=0
MOVL C00458 V=800.0 PL=0
MOVL C00459 V=800.0 PL=0
MOVL C00460 V=800.0 PL=0
MOVL C00461 V=800.0 PL=0
MOVL C00462 V=800.0 PL=0
MOVL C00463 V=800.0 PL=0
MOVL C00464 V=800.0 PL=0
MOVL C00465 V=800.0 PL=0
MOVL C00466 V=800.0 PL=0
MOVL C00467 V=800.0 PL=0
MOVL C00468 V=800.0 PL=0
MOVL C00469 V=800.0 PL=0
MOVL C00470 V=800.0 PL=0
MOVL C00471 V=800.0 PL=0
MOVL C00472 V=800.0 PL=0
MOVL C00473 V=800.0 PL=0
MOVL C00474 V=800.0 PL=0
MOVL C00475 V=800.0 PL=0
MOVL C00476 V=800.0 PL=0
MOVL C00477 V=800.0 PL=0
MOVL C00478 V=800.0 PL=0
MOVL C00479 V=800.0 PL=0
MOVL C00480 V=800.0 PL=0
MOVL C00481 V=800.0 PL=0
MOVL C00482 V=800.0 PL=0
MOVL C00483 V=800.0 PL=0
MOVL C00484 V=800.0 PL=0
MOVL C00485 V=800.0 PL=0
MOVL C00486 V=800.0 PL=0
MOVL C00487 V=800.0 PL=0
MOVL C00488 V=800.0 PL=0
MOVL C00489 V=800.0 PL=0
MOVL C00490 V=800.0 PL=0
MOVL C00491 V=800.0 PL=0
MOVL C00492 V=800.0 PL=0
MOVL C00493 V=800.0 PL=0
MOVL C00494 V=800.0 PL=0
MOVL C00495 V=800.0 PL=0
MOVL C00496 V=800.0 PL=0
MOVL C00497 V=800.0 PL=0
MOVL C00498 V=800.0 PL=0
MOVL C00499 V=800.0 PL=0
MOVL C00500 V=800.0 PL=0
MOVL C00501 V=800.0 PL=0
MOVL C00502 V=800.0 PL=0
MOVL C00503 V=800.0 PL=0
MOVL C00504 V=800.0 PL=0
MOVL C00505 V=800.0 PL=0
MOVL C00506 V=800.0 PL=0
MOVL C00507 V=800.0 PL=0
MOVL C00508 V=800.0 PL=0
MOVL C00509 V=800.0 PL=0
MOVL C00510 V=800.0 PL=0
MOVL C00511 V=800.0 PL=0
MOVL C00512 V=800.0 PL=0
MOVL C00513 V=800.0 PL=0
MOVL C00514 V=800.0 PL=0
MOVL C00515 V=800.0 PL=0
MOVL C00516 V=800.0 PL=0
MOVL C00517 V=800.0 PL=0
MOVL C00518 V=800.0 PL=0
MOVL C00519 V=800.0 PL=0
MOVL C00520 V=800.0 PL=0
MOVL C00521 V=800.0 PL=0
MOVL C00522 V=800.0 PL=0
MOVL C00523 V=800.0 PL=0
MOVL C00524 V=800.0 PL=0
MOVL C00525 V=800.0 PL=0
MOVL C00526 V=800.0 PL=0
MOVL C00527 V=800.0 PL=0
MOVL C00528 V=800.0 PL=0
MOVL C00529 V=800.0 PL=0
MOVL C00530 V=800.0 PL=0
MOVL C00531 V=800.0 PL=0
MOVL C00532 V=800.0 PL=0
MOVL C00533 V=800.0 PL=0
MOVL C00534 V=800.0 PL=0
MOVL C00535 V=800.0 PL=0
MOVL C00536 V=800.0 PL=0
MOVL C00537 V=800.0 PL=0
MOVL C00538 V=800.0 PL=0
MOVL C00539 V=800.0 PL=0
MOVL C00540 V=800.0 PL=0
MOVL C00541 V=800.0 PL=0
MOVL C00542 V=800.0 PL=0
MOVL C00543 V=800.0 PL=0
MOVL C00544 V=800.0 PL=0
MOVL C00545 V=800.0 PL=0
MOVL C00546 V=800.0 PL=0
MOVL C00547 V=800.0 PL=0
MOVL C00548 V=800.0 PL=0
MOVL C00549 V=800.0 PL=0
MOVL C00550 V=800.0 PL=0
MOVL C00551 V=800.0 PL=0
MOVL C00552 V=800.0 PL=0
MOVL C00553 V=800.0 PL=0
MOVL C00554 V=800.0 PL=0
MOVL C00555 V=800.0 PL=0
MOVL C00556 V=800.0 PL=0
MOVL C00557 V=800.0 PL=0
MOVL C00558 V=800.0 PL=0
MOVL C00559 V=800.0 PL=0
MOVL C00560 V=800.0 PL=0
MOVL C00561 V=800.0 PL=0
MOVL C00562 V=800.0 PL=0
MOVL C00563 V=800.0 PL=0
MOVL C00564 V=800.0 PL=0
MOVL C00565 V=800.0 PL=0
MOVL C00566 V=800.0 PL=0
MOVL C00567 V=800.0 PL=0
MOVL C00568 V=800.0 PL=0
MOVL C00569 V=800.0 PL=0
MOVL C00570 V=800.0 PL=0
MOVL C00571 V=800.0 PL=0
MOVL C00572 V=800.0 PL=0
MOVL C00573 V=800.0 PL=0
MOVL C00574 V=800.0 PL=0
MOVL C00575 V=800.0 PL=0
MOVL C00576 V=800.0 PL=0
MOVL C00577 V=800.0 PL=0
MOVL C00578 V=800.0 PL=0
MOVL C00579 V=800.0 PL=0
MOVL C00580 V=800.0 PL=0
MOVL C00581 V=800.0 PL=0
MOVL C00582 V=800.0 PL=0
MOVL C00583 V=800.0 PL=0
MOVL C00584 V=800.0 PL=0
MOVL C00585 V=800.0 PL=0
MOVL C00586 V=800.0 PL=0
MOVL C00587 V=800.0 PL=0
MOVL C00588 V=800.0 PL=0
MOVL C00589 V=800.0 PL=0
MOVL C00590 V=800.0 PL=0
MOVL C00591 V=800.0 PL=0
MOVL C00592 V=800.0 PL=0
MOVL C00593 V=800.0 PL=0
MOVL C00594 V=800.0 PL=0
MOVL C00595 V=800.0 PL=0
MOVL C00596 V=800.0 PL=0
MOVL C00597 V=800.0 PL=0
MOVL C00598 V=800.0 PL=0
MOVL C00599 V=800.0 PL=0
MOVL C00600 V=800.0 PL=0
MOVL C00601 V=800.0 PL=0
MOVL C00602 V=800.0 PL=0
MOVL C00603 V=800.0 PL=0
MOVL C00604 V=800.0 PL=0
MOVL C00605 V=800.0 PL=0
MOVL C00606 V=800.0 PL=0
MOVL C00607 V=800.0 PL=0
MOVL C00608 V=800.0 PL=0
MOVL C00609 V=800.0 PL=0
MOVL C00610 V=800.0 PL=0
MOVL C00611 V=800.0 PL=0
MOVL C00612 V=800.0 PL=0
MOVL C00613 V=800.0 PL=0
MOVL C00614 V=800.0 PL=0
MOVL C00615 V=800.0 PL=0
MOVL C00616 V=800.0 PL=0
MOVL C00617 V=800.0 PL=0
MOVL C00618 V=800.0 PL=0
MOVL C00619 V=800.0 PL=0
MOVL C00620 V=800.0 PL=0
MOVL C00621 V=800.0 PL=0
MOVL C00622 V=800.0 PL=0
MOVL C00623 V=800.0 PL=0
MOVL C00624 V=800.0 PL=0
MOVL C00625 V=800.0 PL=0
MOVL C00626 V=800.0 PL=0
MOVL C00627 V=800.0 PL=0
MOVL C00628 V=800.0 PL=0
MOVL C00629 V=800.0 PL=0
MOVL C00630 V=800.0 PL=0
MOVL C00631 V=800.0 PL=0
MOVL C00632 V=800.0 PL=0
MOVL C00633 V=800.0 PL=0
MOVL C00634 V=800.0 PL=0
MOVL C00635 V=800.0 PL=0
MOVL C00636 V=800.0 PL=0
MOVL C00637 V=800.0 PL=0
MOVL C00638 V=800.0 PL=0
MOVL C00639 V=800.0 PL=0
MOVL C00640 V=800.0 PL=0
MOVL C00641 V=800.0 PL=0
MOVL C00642 V=800.0 PL=0
MOVL C00643 V=800.0 PL=0
MOVL C00644 V=800.0 PL=0
MOVL C00645 V=800.0 PL=0
MOVL C00646 V=800.0 PL=0
MOVL C00647 V=800.0 PL=0
MOVL C00648 V=800.0 PL=0
MOVL C00649 V=800.0 PL=0
MOVL C00650 V=800.0 PL=0
MOVL C00651 V=800.0 PL=0
MOVL C00652 V=800.0 PL=0
MOVL C00653 V=800.0 PL=0
MOVL C00654 V=800.0 PL=0
MOVL C00655 V=800.0 PL=0
MOVL C00656 V=800.0 PL=0
MOVL C00657 V=800.0 PL=0
MOVL C00658 V=800.0 PL=0
MOVL C00659 V=800.0 PL=0
MOVL C00660 V=800.0 PL=0
MOVL C00661 V=800.0 PL=0
MOVL C00662 V=800.0 PL=0
MOVL C00663 V=800.0 PL=0
MOVL C00664 V=800.0 PL=0
MOVL C00665 V=800.0 PL=0
MOVL C00666 V=800.0 PL=0
MOVL C00667 V=800.0 PL=0
MOVL C00668 V=800.0 PL=0
MOVL C00669 V=800.0 PL=0
MOVL C00670 V=800.0 PL=0
MOVL C00671 V=800.0 PL=0
MOVL C00672 V=800.0 PL=0
MOVL C00673 V=800.0 PL=0
MOVL C00674 V=800.0 PL=0
MOVL C00675 V=800.0 PL=0
MOVL C00676 V=800.0 PL=0
MOVL C00677 V=800.0 PL=0
MOVL C00678 V=800.0 PL=0
MOVL C00679 V=800.0 PL=0
MOVL C00680 V=800.0 PL=0
MOVL C00681 V=800.0 PL=0
MOVL C00682 V=800.0 PL=0
MOVL C00683 V=800.0 PL=0
MOVL C00684 V=800.0 PL=0
MOVL C00685 V=800.0 PL=0
MOVL C00686 V=800.0 PL=0
MOVL C00687 V=800.0 PL=0
MOVL C00688 V=800.0 PL=0
MOVL C00689 V=800.0 PL=0
MOVL C00690 V=800.0 PL=0
MOVL C00691 V=800.0 PL=0
MOVL C00692 V=800.0 PL=0
MOVL C00693 V=800.0 PL=0
MOVL C00694 V=800.0 PL=0
MOVL C00695 V=800.0 PL=0
MOVL C00696 V=800.0 PL=0
MOVL C00697 V=800.0 PL=0
MOVL C00698 V=800.0 PL=0
MOVL C00699 V=800.0 PL=0
MOVL C00700 V=800.0 PL=0
MOVL C00701 V=800.0 PL=0
MOVL C00702 V=800.0 PL=0
MOVL C00703 V=800.0 PL=0
MOVL C00704 V=800.0 PL=0
MOVL C00705 V=800.0 PL=0
MOVL C00706 V=800.0 PL=0
MOVL C00707 V=800.0 PL=0
MOVL C00708 V=800.0 PL=0
MOVL C00709 V=800.0 PL=0
MOVL C00710 V=800.0 PL=0
MOVL C00711 V=800.0 PL=0
MOVL C00712 V=800.0 PL=0
MOVL C00713 V=800.0 PL=0
MOVL C00714 V=800.0 PL=0
MOVL C00715 V=800.0 PL=0
MOVL C00716 V=800.0 PL=0
MOVL C00717 V=800.0 PL=0
MOVL C00718 V=800.0 PL=0
MOVL C00719 V=800.0 PL=0
MOVL C00720 V=800.0 PL=0
MOVL C00721 V=800.0 PL=0
MOVL C00722 V=800.0 PL=0
MOVL C00723 V=800.0 PL=0
MOVL C00724 V=800.0 PL=0
MOVL C00725 V=800.0 PL=0
MOVL C00726 V=800.0 PL=0
MOVL C00727 V=800.0 PL=0
MOVL C00728 V=800.0 PL=0
MOVL C00729 V=800.0 PL=0
MOVL C00730 V=800.0 PL=0
MOVL C00731 V=800.0 PL=0
MOVL C00732 V=800.0 PL=0
MOVL C00733 V=800.0 PL=0
MOVL C00734 V=800.0 PL=0
MOVL C00735 V=800.0 PL=0
MOVL C00736 V=800.0 PL=0
MOVL C00737 V=800.0 PL=0
MOVL C00738 V=800.0 PL=0
MOVL C00739 V=800.0 PL=0
MOVL C00740 V=800.0 PL=0
MOVL C00741 V=800.0 PL=0
MOVL C00742 V=800.0 PL=0
MOVL C00743 V=800.0 PL=0
MOVL C00744 V=800.0 PL=0
MOVL C00745 V=800.0 PL=0
MOVL C00746 V=800.0 PL=0
MOVL C00747 V=800.0 PL=0
MOVL C00748 V=800.0 PL=0
MOVL C00749 V=800.0 PL=0
MOVL C00750 V=800.0 PL=0
MOVL C00751 V=800.0 PL=0
MOVL C00752 V=800.0 PL=0
MOVL C00753 V=800.0 PL=0
MOVL C00754 V=800.0 PL=0
MOVL C00755 V=800.0 PL=0
MOVL C00756 V=800.0 PL=0
MOVL C00757 V=800.0 PL=0
MOVL C00758 V=800.0 PL=0
MOVL C00759 V=800.0 PL=0
MOVL C00760 V=800.0 PL=0
MOVL C00761 V=800.0 PL=0
MOVL C00762 V=800.0 PL=0
MOVL C00763 V=800.0 PL=0
MOVL C00764 V=800.0 PL=0
MOVL C00765 V=800.0 PL=0
MOVL C00766 V=800.0 PL=0
MOVL C00767 V=800.0 PL=0
MOVL C00768 V=800.0 PL=0
MOVL C00769 V=800.0 PL=0
MOVL C00770 V=800.0 PL=0
MOVL C00771 V=800.0 PL=0
MOVL C00772 V=800.0 PL=0
MOVL C00773 V=800.0 PL=0
MOVL C00774 V=800.0 PL=0
MOVL C00775 V=800.0 PL=0
MOVL C00776 V=800.0 PL=0
MOVL C00777 V=800.0 PL=0
MOVL C00778 V=800.0 PL=0
MOVL C00779 V=800.0 PL=0
MOVL C00780 V=800.0 PL=0
MOVL C00781 V=800.0 PL=0
MOVL C00782 V=800.0 PL=0
MOVL C00783 V=800.0 PL=0
MOVL C00784 V=800.0 PL=0
MOVL C00785 V=800.0 PL=0
MOVL C00786 V=800.0 PL=0
MOVL C00787 V=800.0 PL=0
MOVL C00788 V=800.0 PL=0
MOVL C00789 V=800.0 PL=0
MOVL C00790 V=800.0 PL=0
MOVL C00791 V=800.0 PL=0
MOVL C00792 V=800.0 PL=0
MOVL C00793 V=800.0 PL=0
MOVL C00794 V=800.0 PL=0
MOVL C00795 V=800.0 PL=0
MOVL C00796 V=800.0 PL=0
MOVL C00797 V=800.0 PL=0
MOVL C00798 V=800.0 PL=0
MOVL C00799 V=800.0 PL=0
MOVL C00800 V=800.0 PL=0
MOVL C00801 V=800.0 PL=0
MOVL C00802 V=800.0 PL=0
MOVL C00803 V=800.0 PL=0
MOVL C00804 V=800.0 PL=0
MOVL C00805 V=800.0 PL=0
MOVL C00806 V=800.0 PL=0
MOVL C00807 V=800.0 PL=0
MOVL C00808 V=800.0 PL=0
MOVL C00809 V=800.0 PL=0
MOVL C00810 V=800.0 PL=0
MOVL C00811 V=800.0 PL=0
MOVL C00812 V=800.0 PL=0
MOVL C00813 V=800.0 PL=0
MOVL C00814 V=800.0 PL=0
MOVL C00815 V=800.0 PL=0
MOVL C00816 V=800.0 PL=0
MOVL C00817 V=800.0 PL=0
MOVL C00818 V=800.0 PL=0
MOVL C00819 V=800.0 PL=0
MOVL C00820 V=800.0 PL=0
MOVL C00821 V=800.0 PL=0
MOVL C00822 V=800.0 PL=0
MOVL C00823 V=800.0 PL=0
MOVL C00824 V=800.0 PL=0
MOVL C00825 V=800.0 PL=0
MOVL C00826 V=800.0 PL=0
MOVL C00827 V=800.0 PL=0
MOVL C00828 V=800.0 PL=0
MOVL C00829 V=800.0 PL=0
MOVL C00830 V=800.0 PL=0
MOVL C00831 V=800.0 PL=0
MOVL C00832 V=800.0 PL=0
MOVL C00833 V=800.0 PL=0
MOVL C00834 V=800.0 PL=0
MOVL C00835 V=800.0 PL=0
MOVL C00836 V=800.0 PL=0
MOVL C00837 V=800.0 PL=0
MOVL C00838 V=800.0 PL=0
MOVL C00839 V=800.0 PL=0
MOVL C00840 V=800.0 PL=0
MOVL C00841 V=800.0 PL=0
MOVL C00842 V=800.0 PL=0
MOVL C00843 V=800.0 PL=0
MOVL C00844 V=800.0 PL=0
MOVL C00845 V=800.0 PL=0
MOVL C00846 V=800.0 PL=0
MOVL C00847 V=800.0 PL=0
MOVL C00848 V=800.0 PL=0
MOVL C00849 V=800.0 PL=0
MOVL C00850 V=800.0 PL=0
MOVL C00851 V=800.0 PL=0
MOVL C00852 V=800.0 PL=0
MOVL C00853 V=800.0 PL=0
MOVL C00854 V=800.0 PL=0
MOVL C00855 V=800.0 PL=0
MOVL C00856 V=800.0 PL=0
MOVL C00857 V=800.0 PL=0
MOVL C00858 V=800.0 PL=0
MOVL C00859 V=800.0 PL=0
MOVL C00860 V=800.0 PL=0
MOVL C00861 V=800.0 PL=0
MOVL C00862 V=800.0 PL=0
MOVL C00863 V=800.0 PL=0
MOVL C00864 V=800.0 PL=0
MOVL C00865 V=800.0 PL=0
MOVL C00866 V=800.0 PL=0
MOVL C00867 V=800.0 PL=0
MOVL C00868 V=800.0 PL=0
MOVL C00869 V=800.0 PL=0
MOVL C00870 V=800.0 PL=0
MOVL C00871 V=800.0 PL=0
MOVL C00872 V=800.0 PL=0
MOVL C00873 V=800.0 PL=0
MOVL C00874 V=800.0 PL=0
MOVL C00875 V=800.0 PL=0
MOVL C00876 V=800.0 PL=0
MOVL C00877 V=800.0 PL=0
MOVL C00878 V=800.0 PL=0
MOVL C00879 V=800.0 PL=0
MOVL C00880 V=800.0 PL=0
MOVL C00881 V=800.0 PL=0
MOVL C00882 V=800.0 PL=0
MOVL C00883 V=800.0 PL=0
MOVL C00884 V=800.0 PL=0
MOVL C00885 V=800.0 PL=0
MOVL C00886 V=800.0 PL=0
MOVL C00887 V=800.0 PL=0
MOVL C00888 V=800.0 PL=0
MOVL C00889 V=800.0 PL=0
MOVL C00890 V=800.0 PL=0
MOVL C00891 V=800.0 PL=0
MOVL C00892 V=800.0 PL=0
MOVL C00893 V=800.0 PL=0
MOVL C00894 V=800.0 PL=0
MOVL C00895 V=800.0 PL=0
MOVL C00896 V=800.0 PL=0
MOVL C00897 V=800.0 PL=0
MOVL C00898 V=800.0 PL=0
MOVL C00899 V=800.0 PL=0
MOVL C00900 V=800.0 PL=0
MOVL C00901 V=800.0 PL=0
MOVL C00902 V=800.0 PL=0
MOVL C00903 V=800.0 PL=0
MOVL C00904 V=800.0 PL=0
MOVL C00905 V=800.0 PL=0
MOVL C00906 V=800.0 PL=0
MOVL C00907 V=800.0 PL=0
MOVL C00908 V=800.0 PL=0
MOVL C00909 V=800.0 PL=0
MOVL C00910 V=800.0 PL=0
MOVL C00911 V=800.0 PL=0
MOVL C00912 V=800.0 PL=0
MOVL C00913 V=800.0 PL=0
MOVL C00914 V=800.0 PL=0
MOVL C00915 V=800.0 PL=0
MOVL C00916 V=800.0 PL=0
MOVL C00917 V=800.0 PL=0
MOVL C00918 V=800.0 PL=0
MOVL C00919 V=800.0 PL=0
MOVL C00920 V=800.0 PL=0
MOVL C00921 V=800.0 PL=0
MOVL C00922 V=800.0 PL=0
MOVL C00923 V=800.0 PL=0
MOVL C00924 V=800.0 PL=0
MOVL C00925 V=800.0 PL=0
MOVL C00926 V=800.0 PL=0
MOVL C00927 V=800.0 PL=0
MOVL C00928 V=800.0 PL=0
MOVL C00929 V=800.0 PL=0
MOVL C00930 V=800.0 PL=0
MOVL C00931 V=800.0 PL=0
MOVL C00932 V=800.0 PL=0
MOVL C00933 V=800.0 PL=0
MOVL C00934 V=800.0 PL=0
MOVL C00935 V=800.0 PL=0
MOVL C00936 V=800.0 PL=0
MOVL C00937 V=800.0 PL=0
MOVL C00938 V=800.0 PL=0
MOVL C00939 V=800.0 PL=0
MOVL C00940 V=800.0 PL=0
MOVL C00941 V=800.0 PL=0
MOVL C00942 V=800.0 PL=0
MOVL C00943 V=800.0 PL=0
MOVL C00944 V=800.0 PL=0
MOVL C00945 V=800.0 PL=0
MOVL C00946 V=800.0 PL=0
MOVL C00947 V=800.0 PL=0
MOVL C00948 V=800.0 PL=0
MOVL C00949 V=800.0 PL=0
MOVL C00950 V=800.0 PL=0
MOVL C00951 V=800.0 PL=0
MOVL C00952 V=800.0 PL=0
MOVL C00953 V=800.0 PL=0
MOVL C00954 V=800.0 PL=0
MOVL C00955 V=800.0 PL=0
MOVL C00956 V=800.0 PL=0
MOVL C00957 V=800.0 PL=0
MOVL C00958 V=800.0 PL=0
MOVL C00959 V=800.0 PL=0
MOVL C00960 V=800.0 PL=0
MOVL C00961 V=800.0 PL=0
MOVL C00962 V=800.0 PL=0
MOVL C00963 V=800.0 PL=0
MOVL C00964 V=800.0 PL=0
MOVL C00965 V=800.0 PL=0
MOVL C00966 V=800.0 PL=0
MOVL C00967 V=800.0 PL=0
MOVL C00968 V=800.0 PL=0
MOVL C00969 V=800.0 PL=0
MOVL C00970 V=800.0 PL=0
MOVL C00971 V=800.0 PL=0
MOVL C00972 V=800.0 PL=0
MOVL C00973 V=800.0 PL=0
MOVL C00974 V=800.0 PL=0
MOVL C00975 V=800.0 PL=0
MOVL C00976 V=800.0 PL=0
MOVL C00977 V=800.0 PL=0
MOVL C00978 V=800.0 PL=0
MOVL C00979 V=800.0 PL=0
MOVL C00980 V=800.0 PL=0
MOVL C00981 V=800.0 PL=0
MOVL C00982 V=800.0 PL=0
MOVL C00983 V=800.0 PL=0
MOVL C00984 V=800.0 PL=0
MOVL C00985 V=800.0 PL=0
MOVL C00986 V=800.0 PL=0
MOVL C00987 V=800.0 PL=0
MOVL C00988 V=800.0 PL=0
MOVL C00989 V=800.0 PL=0
MOVL C00990 V=800.0 PL=0
MOVL C00991 V=800.0 PL=0
MOVL C00992 V=800.0 PL=0
MOVL C00993 V=800.0 PL=0
MOVL C00994 V=800.0 PL=0
MOVL C00995 V=800.0 PL=0
MOVL C00996 V=800.0 PL=0
MOVL C00997 V=800.0 PL=0
MOVL C00998 V=800.0 PL=0
MOVL C00999 V=800.0 PL=0
MOVL C01000 V=800.0 PL=0
MOVL C01001 V=800.0 PL=0
MOVL C01002 V=800.0 PL=0
MOVL C01003 V=800.0 PL=0
MOVL C01004 V=800.0 PL=0
MOVL C01005 V=800.0 PL=0
MOVL C01006 V=800.0 PL=0
MOVL C01007 V=800.0 PL=0
MOVL C01008 V=800.0 PL=0
MOVL C01009 V=800.0 PL=0
MOVL C01010 V=800.0 PL=0
MOVL C01011 V=800.0 PL=0
MOVL C01012 V=800.0 PL=0
MOVL C01013 V=800.0 PL=0
MOVL C01014 V=800.0 PL=0
MOVL C01015 V=800.0 PL=0
MOVL C01016 V=800.0 PL=0
MOVL C01017 V=800.0 PL=0
MOVL C01018 V=800.0 PL=0
MOVL C01019 V=800.0 PL=0
MOVL C01020 V=800.0 PL=0
MOVL C01021 V=800.0 PL=0
MOVL C01022 V=800.0 PL=0
MOVL C01023 V=800.0 PL=0
MOVL C01024 V=800.0 PL=0
MOVL C01025 V=800.0 PL=0
MOVL C01026 V=800.0 PL=0
MOVL C01027 V=800.0 PL=0
MOVL C01028 V=800.0 PL=0
MOVL C01029 V=800.0 PL=0
MOVL C01030 V=800.0 PL=0
MOVL C01031 V=800.0 PL=0
MOVL C01032 V=800.0 PL=0
MOVL C01033 V=800.0 PL=0
MOVL C01034 V=800.0 PL=0
MOVL C01035 V=800.0 PL=0
MOVL C01036 V=800.0 PL=0
MOVL C01037 V=800.0 PL=0
MOVL C01038 V=800.0 PL=0
MOVL C01039 V=800.0 PL=0
MOVL C01040 V=800.0 PL=0
MOVL C01041 V=800.0 PL=0
MOVL C01042 V=800.0 PL=0
MOVL C01043 V=800.0 PL=0
MOVL C01044 V=800.0 PL=0
MOVL C01045 V=800.0 PL=0
MOVL C01046 V=800.0 PL=0
MOVL C01047 V=800.0 PL=0
MOVL C01048 V=800.0 PL=0
MOVL C01049 V=800.0 PL=0
MOVL C01050 V=800.0 PL=0
MOVL C01051 V=800.0 PL=0
MOVL C01052 V=800.0 PL=0
MOVL C01053 V=800.0 PL=0
MOVL C01054 V=800.0 PL=0
MOVL C01055 V=800.0 PL=0
MOVL C01056 V=800.0 PL=0
MOVL C01057 V=800.0 PL=0
MOVL C01058 V=800.0 PL=0
MOVL C01059 V=800.0 PL=0
MOVL C01060 V=800.0 PL=0
MOVL C01061 V=800.0 PL=0
MOVL C01062 V=800.0 PL=0
MOVL C01063 V=800.0 PL=0
MOVL C01064 V=800.0 PL=0
MOVL C01065 V=800.0 PL=0
MOVL C01066 V=800.0 PL=0
MOVL C01067 V=800.0 PL=0
MOVL C01068 V=800.0 PL=0
MOVL C01069 V=800.0 PL=0
MOVL C01070 V=800.0 PL=0
MOVL C01071 V=800.0 PL=0
MOVL C01072 V=800.0 PL=0
MOVL C01073 V=800.0 PL=0
MOVL C01074 V=800.0 PL=0
MOVL C01075 V=800.0 PL=0
MOVL C01076 V=800.0 PL=0
MOVL C01077 V=800.0 PL=0
MOVL C01078 V=800.0 PL=0
MOVL C01079 V=800.0 PL=0
MOVL C01080 V=800.0 PL=0
MOVL C01081 V=800.0 PL=0
MOVL C01082 V=800.0 PL=0
MOVL C01083 V=800.0 PL=0
MOVL C01084 V=800.0 PL=0
MOVL C01085 V=800.0 PL=0
MOVL C01086 V=800.0 PL=0
MOVL C01087 V=800.0 PL=0
MOVL C01088 V=800.0 PL=0
MOVL C01089 V=800.0 PL=0
MOVL C01090 V=800.0 PL=0
MOVL C01091 V=800.0 PL=0
MOVL C01092 V=800.0 PL=0
MOVL C01093 V=800.0 PL=0
MOVL C01094 V=800.0 PL=0
MOVL C01095 V=800.0 PL=0
MOVL C01096 V=800.0 PL=0
MOVL C01097 V=800.0 PL=0
MOVL C01098 V=800.0 PL=0
MOVL C01099 V=800.0 PL=0
MOVL C01100 V=800.0 PL=0
MOVL C01101 V=800.0 PL=0
MOVL C01102 V=800.0 PL=0
MOVL C01103 V=800.0 PL=0
MOVL C01104 V=800.0 PL=0
MOVL C01105 V=800.0 PL=0
MOVL C01106 V=800.0 PL=0
MOVL C01107 V=800.0 PL=0
MOVL C01108 V=800.0 PL=0
MOVL C01109 V=800.0 PL=0
MOVL C01110 V=800.0 PL=0
MOVL C01111 V=800.0 PL=0
MOVL C01112 V=800.0 PL=0
MOVL C01113 V=800.0 PL=0
MOVL C01114 V=800.0 PL=0
MOVL C01115 V=800.0 PL=0
MOVL C01116 V=800.0 PL=0
MOVL C01117 V=800.0 PL=0
MOVL C01118 V=800.0 PL=0
MOVL C01119 V=800.0 PL=0
MOVL C01120 V=800.0 PL=0
MOVL C01121 V=800.0 PL=0
MOVL C01122 V=800.0 PL=0
MOVL C01123 V=800.0 PL=0
MOVL C01124 V=800.0 PL=0
MOVL C01125 V=800.0 PL=0
MOVL C01126 V=800.0 PL=0
MOVL C01127 V=800.0 PL=0
MOVL C01128 V=800.0 PL=0
MOVL C01129 V=800.0 PL=0
MOVL C01130 V=800.0 PL=0
MOVL C01131 V=800.0 PL=0
MOVL C01132 V=800.0 PL=0
MOVL C01133 V=800.0 PL=0
MOVL C01134 V=800.0 PL=0
MOVL C01135 V=800.0 PL=0
MOVL C01136 V=800.0 PL=0
MOVL C01137 V=800.0 PL=0
MOVL C01138 V=800.0 PL=0
MOVL C01139 V=800.0 PL=0
MOVL C01140 V=800.0 PL=0
MOVL C01141 V=800.0 PL=0
MOVL C01142 V=800.0 PL=0
MOVL C01143 V=800.0 PL=0
MOVL C01144 V=800.0 PL=0
MOVL C01145 V=800.0 PL=0
MOVL C01146 V=800.0 PL=0
MOVL C01147 V=800.0 PL=0
MOVL C01148 V=800.0 PL=0
MOVL C01149 V=800.0 PL=0
MOVL C01150 V=800.0 PL=0
MOVL C01151 V=800.0 PL=0
MOVL C01152 V=800.0 PL=0
MOVL C01153 V=800.0 PL=0
MOVL C01154 V=800.0 PL=0
MOVL C01155 V=800.0 PL=0
MOVL C01156 V=800.0 PL=0
MOVL C01157 V=800.0 PL=0
MOVL C01158 V=800.0 PL=0
MOVL C01159 V=800.0 PL=0
MOVL C01160 V=800.0 PL=0
MOVL C01161 V=800.0 PL=0
MOVL C01162 V=800.0 PL=0
MOVL C01163 V=800.0 PL=0
MOVL C01164 V=800.0 PL=0
MOVL C01165 V=800.0 PL=0
MOVL C01166 V=800.0 PL=0
MOVL C01167 V=800.0 PL=0
MOVL C01168 V=800.0 PL=0
MOVL C01169 V=800.0 PL=0
MOVL C01170 V=800.0 PL=0
MOVL C01171 V=800.0 PL=0
MOVL C01172 V=800.0 PL=0
MOVL C01173 V=800.0 PL=0
MOVL C01174 V=800.0 PL=0
MOVL C01175 V=800.0 PL=0
MOVL C01176 V=800.0 PL=0
MOVL C01177 V=800.0 PL=0
MOVL C01178 V=800.0 PL=0
MOVL C01179 V=800.0 PL=0
MOVL C01180 V=800.0 PL=0
MOVL C01181 V=800.0 PL=0
MOVL C01182 V=800.0 PL=0
MOVL C01183 V=800.0 PL=0
MOVL C01184 V=800.0 PL=0
MOVL C01185 V=800.0 PL=0
MOVL C01186 V=800.0 PL=0
MOVL C01187 V=800.0 PL=0
MOVL C01188 V=800.0 PL=0
MOVL C01189 V=800.0 PL=0
MOVL C01190 V=800.0 PL=0
MOVL C01191 V=800.0 PL=0
MOVL C01192 V=800.0 PL=0
MOVL C01193 V=800.0 PL=0
MOVL C01194 V=800.0 PL=0
MOVL C01195 V=800.0 PL=0
MOVL C01196 V=800.0 PL=0
MOVL C01197 V=800.0 PL=0
MOVL C01198 V=800.0 PL=0
MOVL C01199 V=800.0 PL=0
MOVL C01200 V=800.0 PL=0
MOVL C01201 V=800.0 PL=0
MOVL C01202 V=800.0 PL=0
MOVL C01203 V=800.0 PL=0
MOVL C01204 V=800.0 PL=0
MOVL C01205 V=800.0 PL=0
MOVL C01206 V=800.0 PL=0
MOVL C01207 V=800.0 PL=0
MOVL C01208 V=800.0 PL=0
MOVL C01209 V=800.0 PL=0
MOVL C01210 V=800.0 PL=0
MOVL C01211 V=800.0 PL=0
MOVL C01212 V=800.0 PL=0
MOVL C01213 V=800.0 PL=0
MOVL C01214 V=800.0 PL=0
MOVL C01215 V=800.0 PL=0
MOVL C01216 V=800.0 PL=0
MOVL C01217 V=800.0 PL=0
MOVL C01218 V=800.0 PL=0
MOVL C01219 V=800.0 PL=0
MOVL C01220 V=800.0 PL=0
MOVL C01221 V=800.0 PL=0
MOVL C01222 V=800.0 PL=0
MOVL C01223 V=800.0 PL=0
MOVL C01224 V=800.0 PL=0
MOVL C01225 V=800.0 PL=0
MOVL C01226 V=800.0 PL=0
MOVL C01227 V=800.0 PL=0
MOVL C01228 V=800.0 PL=0
MOVL C01229 V=800.0 PL=0
MOVL C01230 V=800.0 PL=0
MOVL C01231 V=800.0 PL=0
MOVL C01232 V=800.0 PL=0
MOVL C01233 V=800.0 PL=0
MOVL C01234 V=800.0 PL=0
MOVL C01235 V=800.0 PL=0
MOVL C01236 V=800.0 PL=0
MOVL C01237 V=800.0 PL=0
MOVL C01238 V=800.0 PL=0
MOVL C01239 V=800.0 PL=0
MOVL C01240 V=800.0 PL=0
MOVL C01241 V=800.0 PL=0
MOVL C01242 V=800.0 PL=0
MOVL C01243 V=800.0 PL=0
MOVL C01244 V=800.0 PL=0
MOVL C01245 V=800.0 PL=0
MOVL C01246 V=800.0 PL=0
MOVL C01247 V=800.0 PL=0
MOVL C01248 V=800.0 PL=0
MOVL C01249 V=800.0 PL=0
MOVL C01250 V=800.0 PL=0
MOVL C01251 V=800.0 PL=0
MOVL C01252 V=800.0 PL=0
MOVL C01253 V=800.0 PL=0
MOVL C01254 V=800.0 PL=0
MOVL C01255 V=800.0 PL=0
MOVL C01256 V=800.0 PL=0
MOVL C01257 V=800.0 PL=0
MOVL C01258 V=800.0 PL=0
MOVL C01259 V=800.0 PL=0
MOVL C01260 V=800.0 PL=0
MOVL C01261 V=800.0 PL=0
MOVL C01262 V=800.0 PL=0
MOVL C01263 V=800.0 PL=0
MOVL C01264 V=800.0 PL=0
MOVL C01265 V=800.0 PL=0
MOVL C01266 V=800.0 PL=0
MOVL C01267 V=800.0 PL=0
MOVL C01268 V=800.0 PL=0
MOVL C01269 V=800.0 PL=0
MOVL C01270 V=800.0 PL=0
MOVL C01271 V=800.0 PL=0
MOVL C01272 V=800.0 PL=0
MOVL C01273 V=800.0 PL=0
MOVL C01274 V=800.0 PL=0
MOVL C01275 V=800.0 PL=0
MOVL C01276 V=800.0 PL=0
MOVL C01277 V=800.0 PL=0
MOVL C01278 V=800.0 PL=0
MOVL C01279 V=800.0 PL=0
MOVL C01280 V=800.0 PL=0
MOVL C01281 V=800.0 PL=0
MOVL C01282 V=800.0 PL=0
MOVL C01283 V=800.0 PL=0
MOVL C01284 V=800.0 PL=0
MOVL C01285 V=800.0 PL=0
MOVL C01286 V=800.0 PL=0
MOVL C01287 V=800.0 PL=0
MOVL C01288 V=800.0 PL=0
MOVL C01289 V=800.0 PL=0
MOVL C01290 V=800.0 PL=0
MOVL C01291 V=800.0 PL=0
MOVL C01292 V=800.0 PL=0
MOVL C01293 V=800.0 PL=0
MOVL C01294 V=800.0 PL=0
MOVL C01295 V=800.0 PL=0
MOVL C01296 V=800.0 PL=0
MOVL C01297 V=800.0 PL=0
MOVL C01298 V=800.0 PL=0
MOVL C01299 V=800.0 PL=0
MOVL C01300 V=800.0 PL=0
MOVL C01301 V=800.0 PL=0
MOVL C01302 V=800.0 PL=0
MOVL C01303 V=800.0 PL=0
MOVL C01304 V=800.0 PL=0
MOVL C01305 V=800.0 PL=0
MOVL C01306 V=800.0 PL=0
MOVL C01307 V=800.0 PL=0
MOVL C01308 V=800.0 PL=0
MOVL C01309 V=800.0 PL=0
MOVL C01310 V=800.0 PL=0
MOVL C01311 V=800.0 PL=0
MOVL C01312 V=800.0 PL=0
MOVL C01313 V=800.0 PL=0
MOVL C01314 V=800.0 PL=0
MOVL C01315 V=800.0 PL=0
MOVL C01316 V=800.0 PL=0
MOVL C01317 V=800.0 PL=0
MOVL C01318 V=800.0 PL=0
MOVL C01319 V=800.0 PL=0
MOVL C01320 V=800.0 PL=0
MOVL C01321 V=800.0 PL=0
MOVL C01322 V=800.0 PL=0
MOVL C01323 V=800.0 PL=0
MOVL C01324 V=800.0 PL=0
MOVL C01325 V=800.0 PL=0
MOVL C01326 V=800.0 PL=0
MOVL C01327 V=800.0 PL=0
MOVL C01328 V=800.0 PL=0
MOVL C01329 V=800.0 PL=0
MOVL C01330 V=800.0 PL=0
MOVL C01331 V=800.0 PL=0
MOVL C01332 V=800.0 PL=0
MOVL C01333 V=800.0 PL=0
MOVL C01334 V=800.0 PL=0
MOVL C01335 V=800.0 PL=0
MOVL C01336 V=800.0 PL=0
MOVL C01337 V=800.0 PL=0
MOVL C01338 V=800.0 PL=0
MOVL C01339 V=800.0 PL=0
MOVL C01340 V=800.0 PL=0
MOVL C01341 V=800.0 PL=0
MOVL C01342 V=800.0 PL=0
MOVL C01343 V=800.0 PL=0
MOVL C01344 V=800.0 PL=0
MOVL C01345 V=800.0 PL=0
MOVL C01346 V=800.0 PL=0
MOVL C01347 V=800.0 PL=0
MOVL C01348 V=800.0 PL=0
MOVL C01349 V=800.0 PL=0
MOVL C01350 V=800.0 PL=0
MOVL C01351 V=800.0 PL=0
MOVL C01352 V=800.0 PL=0
MOVL C01353 V=800.0 PL=0
MOVL C01354 V=800.0 PL=0
MOVL C01355 V=800.0 PL=0
MOVL C01356 V=800.0 PL=0
MOVL C01357 V=800.0 PL=0
MOVL C01358 V=800.0 PL=0
MOVL C01359 V=800.0 PL=0
MOVL C01360 V=800.0 PL=0
MOVL C01361 V=800.0 PL=0
MOVL C01362 V=800.0 PL=0
MOVL C01363 V=800.0 PL=0
MOVL C01364 V=800.0 PL=0
MOVL C01365 V=800.0 PL=0
MOVL C01366 V=800.0 PL=0
MOVL C01367 V=800.0 PL=0
MOVL C01368 V=800.0 PL=0
MOVL C01369 V=800.0 PL=0
MOVL C01370 V=800.0 PL=0
MOVL C01371 V=800.0 PL=0
MOVL C01372 V=800.0 PL=0
MOVL C01373 V=800.0 PL=0
MOVL C01374 V=800.0 PL=0
MOVL C01375 V=800.0 PL=0
MOVL C01376 V=800.0 PL=0
MOVL C01377 V=800.0 PL=0
MOVL C01378 V=800.0 PL=0
MOVL C01379 V=800.0 PL=0
MOVL C01380 V=800.0 PL=0
MOVL C01381 V=800.0 PL=0
MOVL C01382 V=800.0 PL=0
MOVL C01383 V=800.0 PL=0
MOVL C01384 V=800.0 PL=0
MOVL C01385 V=800.0 PL=0
MOVL C01386 V=800.0 PL=0
MOVL C01387 V=800.0 PL=0
MOVL C01388 V=800.0 PL=0
MOVL C01389 V=800.0 PL=0
MOVL C01390 V=800.0 PL=0
MOVL C01391 V=800.0 PL=0
MOVL C01392 V=800.0 PL=0
MOVL C01393 V=800.0 PL=0
MOVL C01394 V=800.0 PL=0
MOVL C01395 V=800.0 PL=0
MOVL C01396 V=800.0 PL=0
MOVL C01397 V=800.0 PL=0
MOVL C01398 V=800.0 PL=0
MOVL C01399 V=800.0 PL=0
MOVL C01400 V=800.0 PL=0
MOVL C01401 V=800.0 PL=0
MOVL C01402 V=800.0 PL=0
MOVL C01403 V=800.0 PL=0
MOVL C01404 V=800.0 PL=0
MOVL C01405 V=800.0 PL=0
MOVL C01406 V=800.0 PL=0
MOVL C01407 V=800.0 PL=0
MOVL C01408 V=800.0 PL=0
MOVL C01409 V=800.0 PL=0
MOVL C01410 V=800.0 PL=0
MOVL C01411 V=800.0 PL=0
MOVL C01412 V=800.0 PL=0
MOVL C01413 V=800.0 PL=0
MOVL C01414 V=800.0 PL=0
MOVL C01415 V=800.0 PL=0
MOVL C01416 V=800.0 PL=0
MOVL C01417 V=800.0 PL=0
MOVL C01418 V=800.0 PL=0
MOVL C01419 V=800.0 PL=0
MOVL C01420 V=800.0 PL=0
MOVL C01421 V=800.0 PL=0
MOVL C01422 V=800.0 PL=0
MOVL C01423 V=800.0 PL=0
MOVL C01424 V=800.0 PL=0
MOVL C01425 V=800.0 PL=0
MOVL C01426 V=800.0 PL=0
MOVL C01427 V=800.0 PL=0
MOVL C01428 V=800.0 PL=0
MOVL C01429 V=800.0 PL=0
MOVL C01430 V=800.0 PL=0
MOVL C01431 V=800.0 PL=0
MOVL C01432 V=800.0 PL=0
MOVL C01433 V=800.0 PL=0
MOVL C01434 V=800.0 PL=0
MOVL C01435 V=800.0 PL=0
MOVL C01436 V=800.0 PL=0
MOVL C01437 V=800.0 PL=0
MOVL C01438 V=800.0 PL=0
MOVL C01439 V=800.0 PL=0
MOVL C01440 V=800.0 PL=0
MOVL C01441 V=800.0 PL=0
MOVL C01442 V=800.0 PL=0
MOVL C01443 V=800.0 PL=0
MOVL C01444 V=800.0 PL=0
MOVL C01445 V=800.0 PL=0
MOVL C01446 V=800.0 PL=0
MOVL C01447 V=800.0 PL=0
MOVL C01448 V=800.0 PL=0
MOVL C01449 V=800.0 PL=0
MOVL C01450 V=800.0 PL=0
MOVL C01451 V=800.0 PL=0
MOVL C01452 V=800.0 PL=0
MOVL C01453 V=800.0 PL=0
MOVL C01454 V=800.0 PL=0
MOVL C01455 V=800.0 PL=0
MOVL C01456 V=800.0 PL=0
MOVL C01457 V=800.0 PL=0
MOVL C01458 V=800.0 PL=0
MOVL C01459 V=800.0 PL=0
MOVL C01460 V=800.0 PL=0
MOVL C01461 V=800.0 PL=0
MOVL C01462 V=800.0 PL=0
MOVL C01463 V=800.0 PL=0
MOVL C01464 V=800.0 PL=0
MOVL C01465 V=800.0 PL=0
MOVL C01466 V=800.0 PL=0
MOVL C01467 V=800.0 PL=0
MOVL C01468 V=800.0 PL=0
MOVL C01469 V=800.0 PL=0
MOVL C01470 V=800.0 PL=0
MOVL C01471 V=800.0 PL=0
MOVL C01472 V=800.0 PL=0
MOVL C01473 V=800.0 PL=0
MOVL C01474 V=800.0 PL=0
MOVL C01475 V=800.0 PL=0
MOVL C01476 V=800.0 PL=0
MOVL C01477 V=800.0 PL=0
MOVL C01478 V=800.0 PL=0
MOVL C01479 V=800.0 PL=0
MOVL C01480 V=800.0 PL=0
MOVL C01481 V=800.0 PL=0
MOVL C01482 V=800.0 PL=0
MOVL C01483 V=800.0 PL=0
MOVL C01484 V=800.0 PL=0
MOVL C01485 V=800.0 PL=0
MOVL C01486 V=800.0 PL=0
MOVL C01487 V=800.0 PL=0
MOVL C01488 V=800.0 PL=0
MOVL C01489 V=800.0 PL=0
MOVL C01490 V=800.0 PL=0
MOVL C01491 V=800.0 PL=0
MOVL C01492 V=800.0 PL=0
MOVL C01493 V=800.0 PL=0
MOVL C01494 V=800.0 PL=0
MOVL C01495 V=800.0 PL=0
MOVL C01496 V=800.0 PL=0
MOVL C01497 V=800.0 PL=0
MOVL C01498 V=800.0 PL=0
MOVL C01499 V=800.0 PL=0
MOVL C01500 V=800.0 PL=0
MOVL C01501 V=800.0 PL=0
MOVL C01502 V=800.0 PL=0
MOVL C01503 V=800.0 PL=0
MOVL C01504 V=800.0 PL=0
MOVL C01505 V=800.0 PL=0
MOVL C01506 V=800.0 PL=0
MOVL C01507 V=800.0 PL=0
MOVL C01508 V=800.0 PL=0
MOVL C01509 V=800.0 PL=0
MOVL C01510 V=800.0 PL=0
MOVL C01511 V=800.0 PL=0
MOVL C01512 V=800.0 PL=0
MOVL C01513 V=800.0 PL=0
MOVL C01514 V=800.0 PL=0
MOVL C01515 V=800.0 PL=0
MOVL C01516 V=800.0 PL=0
MOVL C01517 V=800.0 PL=0
MOVL C01518 V=800.0 PL=0
MOVL C01519 V=800.0 PL=0
MOVL C01520 V=800.0 PL=0
MOVL C01521 V=800.0 PL=0
MOVL C01522 V=800.0 PL=0
MOVL C01523 V=800.0 PL=0
MOVL C01524 V=800.0 PL=0
MOVL C01525 V=800.0 PL=0
MOVL C01526 V=800.0 PL=0
MOVL C01527 V=800.0 PL=0
MOVL C01528 V=800.0 PL=0
MOVL C01529 V=800.0 PL=0
MOVL C01530 V=800.0 PL=0
MOVL C01531 V=800.0 PL=0
MOVL C01532 V=800.0 PL=0
MOVL C01533 V=800.0 PL=0
MOVL C01534 V=800.0 PL=0
MOVL C01535 V=800.0 PL=0
MOVL C01536 V=800.0 PL=0
MOVL C01537 V=800.0 PL=0
MOVL C01538 V=800.0 PL=0
MOVL C01539 V=800.0 PL=0
MOVL C01540 V=800.0 PL=0
MOVL C01541 V=800.0 PL=0
MOVL C01542 V=800.0 PL=0
MOVL C01543 V=800.0 PL=0
MOVL C01544 V=800.0 PL=0
MOVL C01545 V=800.0 PL=0
MOVL C01546 V=800.0 PL=0
MOVL C01547 V=800.0 PL=0
MOVL C01548 V=800.0 PL=0
MOVL C01549 V=800.0 PL=0
MOVL C01550 V=800.0 PL=0
MOVL C01551 V=800.0 PL=0
MOVL C01552 V=800.0 PL=0
MOVL C01553 V=800.0 PL=0
MOVL C01554 V=800.0 PL=0
MOVL C01555 V=800.0 PL=0
MOVL C01556 V=800.0 PL=0
MOVL C01557 V=800.0 PL=0
MOVL C01558 V=800.0 PL=0
MOVL C01559 V=800.0 PL=0
MOVL C01560 V=800.0 PL=0
MOVL C01561 V=800.0 PL=0
MOVL C01562 V=800.0 PL=0
MOVL C01563 V=800.0 PL=0
MOVL C01564 V=800.0 PL=0
MOVL C01565 V=800.0 PL=0
MOVL C01566 V=800.0 PL=0
MOVL C01567 V=800.0 PL=0
MOVL C01568 V=800.0 PL=0
MOVL C01569 V=800.0 PL=0
MOVL C01570 V=800.0 PL=0
MOVL C01571 V=800.0 PL=0
MOVL C01572 V=800.0 PL=0
MOVL C01573 V=800.0 PL=0
MOVL C01574 V=800.0 PL=0
MOVL C01575 V=800.0 PL=0
MOVL C01576 V=800.0 PL=0
MOVL C01577 V=800.0 PL=0
MOVL C01578 V=800.0 PL=0
MOVL C01579 V=800.0 PL=0
MOVL C01580 V=800.0 PL=0
MOVL C01581 V=800.0 PL=0
MOVL C01582 V=800.0 PL=0
MOVL C01583 V=800.0 PL=0
MOVL C01584 V=800.0 PL=0
MOVL C01585 V=800.0 PL=0
MOVL C01586 V=800.0 PL=0
MOVL C01587 V=800.0 PL=0
MOVL C01588 V=800.0 PL=0
MOVL C01589 V=800.0 PL=0
MOVL C01590 V=800.0 PL=0
MOVL C01591 V=800.0 PL=0
MOVL C01592 V=800.0 PL=0
MOVL C01593 V=800.0 PL=0
MOVL C01594 V=800.0 PL=0
MOVL C01595 V=800.0 PL=0
MOVL C01596 V=800.0 PL=0
MOVL C01597 V=800.0 PL=0
MOVL C01598 V=800.0 PL=0
MOVL C01599 V=800.0 PL=0
MOVL C01600 V=800.0 PL=0
MOVL C01601 V=800.0 PL=0
MOVL C01602 V=800.0 PL=0
MOVL C01603 V=800.0 PL=0
MOVL C01604 V=800.0 PL=0
MOVL C01605 V=800.0 PL=0
MOVL C01606 V=800.0 PL=0
MOVL C01607 V=800.0 PL=0
MOVL C01608 V=800.0 PL=0
MOVL C01609 V=800.0 PL=0
MOVL C01610 V=800.0 PL=0
MOVL C01611 V=800.0 PL=0
MOVL C01612 V=800.0 PL=0
MOVL C01613 V=800.0 PL=0
MOVL C01614 V=800.0 PL=0
MOVL C01615 V=800.0 PL=0
MOVL C01616 V=800.0 PL=0
MOVL C01617 V=800.0 PL=0
MOVL C01618 V=800.0 PL=0
MOVL C01619 V=800.0 PL=0
MOVL C01620 V=800.0 PL=0
MOVL C01621 V=800.0 PL=0
MOVL C01622 V=800.0 PL=0
MOVL C01623 V=800.0 PL=0
MOVL C01624 V=800.0 PL=0
MOVL C01625 V=800.0 PL=0
MOVL C01626 V=800.0 PL=0
MOVL C01627 V=800.0 PL=0
MOVL C01628 V=800.0 PL=0
MOVL C01629 V=800.0 PL=0
MOVL C01630 V=800.0 PL=0
MOVL C01631 V=800.0 PL=0
MOVL C01632 V=800.0 PL=0
MOVL C01633 V=800.0 PL=0
MOVL C01634 V=800.0 PL=0
MOVL C01635 V=800.0 PL=0
MOVL C01636 V=800.0 PL=0
MOVL C01637 V=800.0 PL=0
MOVL C01638 V=800.0 PL=0
MOVL C01639 V=800.0 PL=0
MOVL C01640 V=800.0 PL=0
MOVL C01641 V=800.0 PL=0
MOVL C01642 V=800.0 PL=0
MOVL C01643 V=800.0 PL=0
MOVL C01644 V=800.0 PL=0
MOVL C01645 V=800.0 PL=0
MOVL C01646 V=800.0 PL=0
MOVL C01647 V=800.0 PL=0
MOVL C01648 V=800.0 PL=0
MOVL C01649 V=800.0 PL=0
MOVL C01650 V=800.0 PL=0
MOVL C01651 V=800.0 PL=0
MOVL C01652 V=800.0 PL=0
MOVL C01653 V=800.0 PL=0
MOVL C01654 V=800.0 PL=0
MOVL C01655 V=800.0 PL=0
MOVL C01656 V=800.0 PL=0
MOVL C01657 V=800.0 PL=0
MOVL C01658 V=800.0 PL=0
MOVL C01659 V=800.0 PL=0
MOVL C01660 V=800.0 PL=0
MOVL C01661 V=800.0 PL=0
MOVL C01662 V=800.0 PL=0
MOVL C01663 V=800.0 PL=0
MOVL C01664 V=800.0 PL=0
MOVL C01665 V=800.0 PL=0
MOVL C01666 V=800.0 PL=0
MOVL C01667 V=800.0 PL=0
MOVL C01668 V=800.0 PL=0
MOVL C01669 V=800.0 PL=0
MOVL C01670 V=800.0 PL=0
MOVL C01671 V=800.0 PL=0
MOVL C01672 V=800.0 PL=0
MOVL C01673 V=800.0 PL=0
MOVL C01674 V=800.0 PL=0
MOVL C01675 V=800.0 PL=0
MOVL C01676 V=800.0 PL=0
MOVL C01677 V=800.0 PL=0
MOVL C01678 V=800.0 PL=0
MOVL C01679 V=800.0 PL=0
MOVL C01680 V=800.0 PL=0
MOVL C01681 V=800.0 PL=0
MOVL C01682 V=800.0 PL=0
MOVL C01683 V=800.0 PL=0
MOVL C01684 V=800.0 PL=0
MOVL C01685 V=800.0 PL=0
MOVL C01686 V=800.0 PL=0
MOVL C01687 V=800.0 PL=0
MOVL C01688 V=800.0 PL=0
MOVL C01689 V=800.0 PL=0
MOVL C01690 V=800.0 PL=0
MOVL C01691 V=800.0 PL=0
MOVL C01692 V=800.0 PL=0
MOVL C01693 V=800.0 PL=0
MOVL C01694 V=800.0 PL=0
MOVL C01695 V=800.0 PL=0
